# B&R Automation Studio project RobotComau (part 2)

#### Main.st
```iecst
PROGRAM _INIT
	(* Insert code here *)
	MpRecipeXml_0.MpLink := ADR(gRecipeXml);
	MpRecipeXml_0.Enable := TRUE;

	MpRecipeRegPar_0.MpLink := ADR(gRecipeXml);
	MpRecipeRegPar_0.Enable := TRUE;
	gAimPos;
	ScrewPosible := TRUE;
	ScrewWasherPosible := TRUE;
	WrenchPosible := TRUE;

	MpFileManagerUI_R(MpLink := ADR(gFileManagerUI_R), Enable :=1 , ErrorReset :=0 , UISetup :=MpFileMngSetup , UIConnect :=ADR(MpFileMngConnectR));
	MpFileMngConnectR.DeviceList.DeviceNames[0] := 'RecipeDir';

END_PROGRAM

PROGRAM _CYCLIC
	(* Insert code here *)

	IF clear THEN

		FOR i := 0 TO 13 BY 1 DO
		gAimPos[i] :=0 ;
		END_FOR;
		ScrewPosible := TRUE;
		ScrewWasherPosible := TRUE;
		WrenchPosible := TRUE;
	END_IF

	FOR i := 0 TO 13 BY 1 DO

		IF gAimPos[i]  = 1 THEN
			ScrewPosible := FALSE;
		END_IF
		IF gAimPos[i]  = 2 THEN
			ScrewWasherPosible := FALSE;
		END_IF
		IF gAimPos[i]  = 3 THEN
			ScrewPosible := FALSE;
			ScrewWasherPosible := FALSE;
		END_IF
		IF gAimPos[i]  = 4 THEN
			WrenchPosible := FALSE;
		END_IF
		IF gAimPos[i]  = 5 THEN
			WrenchPosible := FALSE;
			ScrewPosible := FALSE;
		END_IF
		IF gAimPos[i]  = 6 THEN
			WrenchPosible := FALSE;
			ScrewWasherPosible := FALSE;
		END_IF
		IF gAimPos[i]  = 7 THEN
			WrenchPosible := FALSE;
			ScrewPosible := FALSE;
			ScrewWasherPosible := FALSE;
		END_IF

	END_FOR;

	MpRecipeXml_0();
	MpRecipeXml_0.DeviceName := ADR('RecipeDir');
	MpRecipeRegPar_0();
	MpRecipeRegPar_0.PVName := ADR('gAimPos');

	MpRecipeXml_0.FileName := ADR(name);

	MpFileManagerUI_R();
	tabInfo.NumberOfElements := 0;

	IF MpFileMngConnectR.MessageBox.Type = mpFILE_MSG_OK THEN
		messageType := 'OK';
	ELSIF MpFileMngConnectR.MessageBox.Type = mpFILE_MSG_CONFIRM_DELETE THEN
		messageType := 'DELETE';
	ELSIF MpFileMngConnectR.MessageBox.Type = mpFILE_MSG_CONFIRM_OVERWRITE THEN
		messageType := 'OVERWRITE';
	ELSIF MpFileMngConnectR.MessageBox.Type = mpFILE_MSG_BUSY THEN
		messageType := 'BUSY';
	END_IF

	FOR iFile := 0 TO 49 BY 1 DO
		(* create arrays with file properties *)

		IF tabInfo.NumberOfElements >= iFile THEN
			brsmemcpy(ADR(tabInfo.Name[iFile]), ADR(MpFileMngConnectR.File.List.Items[iFile].Name), SIZEOF(tabInfo.Name[iFile]));
			brsmemcpy(ADR(tabInfo.Size[iFile]), ADR(MpFileMngConnectR.File.List.Items[iFile].Size), SIZEOF(tabInfo.Size[iFile]));
			brsmemcpy(ADR(tabInfo.Type[iFile]), ADR(MpFileMngConnectR.File.List.Items[iFile].ItemType), SIZEOF(tabInfo.Type[iFile]));
			brsmemcpy(ADR(tabInfo.LastModified[iFile]), ADR(MpFileMngConnectR.File.List.Items[iFile].LastModified), SIZEOF(tabInfo.LastModified[iFile]));
		END_IF

		IF tabInfo.SelectedRow = iFile THEN
			MpFileMngConnectR.File.List.Items[iFile].IsSelected := TRUE;
			name2 := MpFileMngConnectR.File.List.Items[iFile].Name;
		END_IF
		(* numbers of elements in the table *)
		IF tabInfo.Type[iFile] <> mpFILE_ITEM_TYPE_NONE THEN
			//			tabInfo.NumberOfElements := iFile;
			tabInfo.NumberOfElements := tabInfo.NumberOfElements + 1;
		END_IF
	END_FOR

	tableShowLimit := tabInfo.NumberOfElements - 1;
	tableConfig := '{"specRows": [ {"from":0, "to":';
	brsitoa(tableShowLimit,ADR(tempString));
	brsstrcat(ADR(tableConfig),ADR(tempString));
	brsstrcat(ADR(tableConfig),ADR(', "visible":true}, {"from":'));
	brsitoa(tabInfo.NumberOfElements,ADR(tempString));
	brsstrcat(ADR(tableConfig),ADR(tempString));
	brsstrcat(ADR(tableConfig),ADR(', "to":49, "visible":false}]}'));

	IF PriorytetS = 1 THEN
		Index[0] := 1;
	ELSIF PriorytetSW = 1 THEN
		Index[0] := 2;
	ELSIF PriorytetW = 1 THEN
		Index[0] := 4;
	END_IF

	IF PriorytetS = 2 THEN
		Index[1] := 1;
	ELSIF PriorytetSW = 2 THEN
		Index[1] := 2;
	ELSIF PriorytetW = 2 THEN
		Index[1] := 4;
	END_IF

	IF PriorytetS = 3 THEN
		Index[2] := 1;
	ELSIF PriorytetSW = 3 THEN
		Index[2] := 2;
	ELSIF PriorytetW = 3 THEN
		Index[2] := 4;
	END_IF

	IF PriorytetS = PriorytetSW OR PriorytetS = PriorytetW OR PriorytetSW = PriorytetW OR
		PriorytetS = 0 OR PriorytetSW = 0 OR PriorytetW = 0
		THEN
		Index[0] := 1;
		Index[1] := 2;
		Index[2] := 4;
	END_IF

END_PROGRAM

PROGRAM _EXIT
	(* Insert code here *)

END_PROGRAM
```

### Types.typ
```iecst
TYPE
	Step_typ :
		(
		ROBOTCTRL_DISABLED,
		ROBOTCTRL_POWER,
		ROBOTCTRL_WAIT_POWER,
		ROBOTCTRL_HOME,
		ROBOTCTRL_WAIT_HOME,
		ROBOTCTRL_READY,
		ROBOTCTRL_CALCULATE,
		ROBOTCTRL_CHECK,
		ROBOTCTRL_CALCULATE_P1,
		ROBOTCTRL_CALCULATE_P2,
		ROBOTCTRL_IS_MOVE_NEEDED,
		ROBOTCTRL_MOVE,
		ROBOTCTRL_ERROR_WRONG_AIM,
		ROBOTCTRL_ERROR,
		ROBOTCTRL_STOP,
		ROBOTCTRL_INTERRUPT,
		ROBOTCTRL_INTERRUPTING,
		ROBOTCTRL_CONTINUE,
		ROBOTCTRL_POWER_OFF,
		ROBOTCTRL_COMPLITE,
		ROBOTCTRL_SWAP,
		ROBOTCTRL_SWAP_MOVE,
		ROBOTCTRL_DEMO
		);
END_TYPE
```

### Variables.var
```iecst
VAR
	AimIsGood : BOOL := FALSE;
	cartezianVSjog : BOOL; (*Wybór miedzy sterowaniem we wspólrzednych wewnetrznych - 0 / zewnętrznych - 1 *)
	cmdContinue : BOOL;
	cmdInterrupt : BOOL;
	Demo : INT;
	DemoAimPos : ARRAY[0..13] OF INT; (*(DEMO) Aim poses used in demo *)
	DemoIndex : ARRAY[0..2] OF INT := [1,2,4]; (*(DEMO) Order Of movess*)
	diAck : BOOL; (*(IN AUTO)Resets of Vision system error*)
	diAuto : BOOL; (*Enables Auto mode*)
	diExecute : BOOL; (*(IN AUTO) Starts moving proedure *)
	diManual : BOOL; (*Enables manual mode*)
	diReset : BOOL; (*(IN AUTO)  Resets the procedure *)
	diSemiAuto : BOOL; (*Enables semiAuto mode*)
	diStart : BOOL; (*(IN AUTO) Sets robot ready *)
	diStop : BOOL; (*(IN AUTO) stops the procedure *)
	HelpfulInt : USINT; (*(SWAP) int that helps with assigning values *)
END_VAR
VAR CONSTANT
	IndexSize : INT := 3; (*Amount of diffrent objects *)
END_VAR
VAR
	MpRoboArm6Axis_0 : MpRoboArm6Axis; (*Robot *)
	P1P2_Ok : BOOL := FALSE; (*flag that shows if P1 and P2 was assigned*)
	PackML_State : STRING[80];
	RoboParameters : MpRoboArm6AxisParType; (*Robot Parameters*)
END_VAR
VAR CONSTANT
	SizeOfArray : INT := 13; (*(x+1)  amount of possible pleaces to move objects *)
END_VAR
VAR
	Step : {REDUND_UNREPLICABLE} Step_typ := (0); (*state robot *)
	Step_State : STRING[80];
	VelocityQ : REAL;
	VelocityQ1 : REAL; (*Przypisanie predkosci do parametru 1 w zależnosci od wyboru wspólrzednych*)
	VelocityQ2 : REAL; (*Przypisanie predkosci do parametru 2 w zależnosci od wyboru wspólrzednych*)
	VelocityQ3 : REAL; (*Przypisanie predkosci do parametru 3 w zależnosci od wyboru wspólrzednych*)
	VelocityQ4 : REAL; (*Przypisanie predkosci do parametru 4 w zależnosci od wyboru wspólrzednych*)
	VelocityQ5 : REAL; (*Przypisanie predkosci do parametru 5 w zależnosci od wyboru wspólrzednych*)
	VelocityQ6 : REAL; (*Przypisanie predkosci do parametru 6 w zależnosci od wyboru wspólrzednych*)
	VisionCalcDone : BOOL;
	SwapStep : USINT := 0; (*(SWAP) used in swap procedure *)
	x : INT := 0;
	VelocityQQ : REAL;
END_VAR
```

### Program Logical/Robot/PackML/PackML_Auto

#### Variables.var
```iecst
VAR
	NotFirstFlag : BOOL;
END_VAR
```

#### Aborted.st
```iecst
ACTION Aborted:

	IF MpPackMLStateIsActive(gPackMLCore,
		mpPACKML_STATE_ABORTED,
		1) THEN

		PackML_State := 'ABORTED';
		MpRoboArm6Axis_0.Power := FALSE;

		IF MpRoboArm6Axis_0.ErrorReset THEN
			MpPackMLStateComplete(gPackMLCore, 1);

			MpPackMLMode_Auto.Clear := 1;

		END_IF;
	END_IF

END_ACTION
```

#### Aborting.st
```iecst
ACTION Aborting:

	IF MpPackMLStateIsActive(gPackMLCore,
		mpPACKML_STATE_ABORTING,
		1) THEN

		MpPackMLMode_Auto.Abort := 0;

		PackML_State := 'ABORTING';
		MpRoboArm6Axis_0.Power := FALSE;

		IF NOT MpRoboArm6Axis_0.PowerOn THEN
			MpPackMLStateComplete(gPackMLCore, 1);

//			Step := ROBOTCTRL_POWER_OFF;
//			Step_State := 'POWER_OFF';

		END_IF;
	END_IF

END_ACTION
```

#### Clearing.st
```iecst
ACTION Clearing:

	IF MpPackMLStateIsActive(gPackMLCore,
		mpPACKML_STATE_CLEARING,
		1) THEN

		MpPackMLMode_Auto.Clear := 0;
		PackML_State := 'CLEARING';

		IF NOT MpRoboArm6Axis_0.Error THEN
			MpPackMLStateComplete(gPackMLCore, 1);

		END_IF;
	END_IF
END_ACTION
```

#### Complete.st
```iecst
ACTION Complete:
	IF MpPackMLStateIsActive(gPackMLCore,
		mpPACKML_STATE_COMPLETE,
		1) THEN

		PackML_State := 'COMPLETE';
		gCompliteFlag:=TRUE;
		//MpPackMLMode_Auto.Stop := 1;

		IF diReset THEN
			MpPackMLStateComplete(gPackMLCore, 1);
			MpPackMLMode_Auto.Reset := 1;
			Step := ROBOTCTRL_POWER;

			//			Step_State := 'POWER';

			END_IF;
	END_IF

END_ACTION
```

#### Completing.st
```iecst
ACTION Completing:
	IF MpPackMLStateIsActive(gPackMLCore,
		mpPACKML_STATE_COMPLETING,
		1) THEN
			PackML_State := 'COMPLETING';
		emptyPos:=0;
			MpPackMLStateComplete(gPackMLCore, 1);

	END_IF

END_ACTION
```

#### Execute.st
```iecst
//   General conception of this code
//  assainging binary values to each object
//	screw      -001 - 1
//  screw pad  -010 - 2
//  wrench     -100 - 4
//  therefore we can assing to gAimPose table values from 0-7 ( sum must equal 7) in order to
//  easly differentiate what kind of object we need to move into aim pose.
//  for example if we see 6 -> 110 we know that we have to move screw pad and wrench to this pose
//
//  order of moves is defined by order of numbers in Index

ACTION Execute:
	IF MpPackMLStateIsActive(gPackMLCore,
		mpPACKML_STATE_EXECUTE,
		1) THEN

		PackML_State := 'EXECUTE';

		CASE Step OF

			ROBOTCTRL_CALCULATE:
				//Reseting buffor
				//blocks which can be used as buffor
				FOR x:=0 TO SizeOfArray DO
					IF  gActPos[x]=0 THEN
						gSwapEnable[x]:=FALSE;
					ELSE
						gSwapEnable[x]:=TRUE;
					END_IF;
				END_FOR;

				IF diDemo THEN
					IF NOT NotFirstFlag THEN
						FOR x:=0 TO SizeOfArray DO
							gDemoActPos[x]:=gActPos[x];
						END_FOR;
					END_IF;

					FOR x:=0 TO SizeOfArray DO
						IF  gDemoActPos[x]=0 AND gIsPosGood[x] THEN
							gPosBuffor[x]:=TRUE;
						ELSE
							gPosBuffor[x]:=FALSE;
						END_IF;
					END_FOR;
				ELSE
					FOR x:=0 TO SizeOfArray DO
						IF  gActPos[x]=0 AND gIsPosGood[x] THEN
							gPosBuffor[x]:=TRUE;
						ELSE
							gPosBuffor[x]:=FALSE;
						END_IF;
					END_FOR;

				END_IF;

				IF diDemo AND NOT P1P2_Ok AND y=0 THEN
					CASE Demo OF

						0:
							DemoY:=0;
							DemoIndex[0]:=1;
							DemoIndex[1]:=2;
							DemoIndex[2]:=4;
							FOR x:=0 TO SizeOfArray DO
								IF DemoY <IndexSize THEN
									IF gPosBuffor[x] THEN
										DemoAimPos[x]:=DemoIndex[DemoY];
										DemoY:=DemoY+1;
									ELSE
										DemoAimPos[x]:=0;

									END_IF;
								ELSE
									DemoAimPos[x]:=0;
								END_IF;
							END_FOR;
							Step:=ROBOTCTRL_CALCULATE_P1;
							Demo:=1;

						1:

							DemoY:=0;
							DemoIndex[0]:=2;
							DemoIndex[1]:=1;
							DemoIndex[2]:=4;
							FOR x:=SizeOfArray TO 0 BY -1 DO
								IF DemoY <IndexSize THEN
									IF gPosBuffor[x] THEN
										DemoAimPos[x]:=DemoIndex[DemoY];
										DemoY:=DemoY+1;
									ELSE
										DemoAimPos[x]:=0;

									END_IF;
								ELSE
									DemoAimPos[x]:=0;
								END_IF;

							END_FOR;
							Step:=ROBOTCTRL_CALCULATE_P1;
							Demo:=2;

						2:

							DemoY:=0;
							DemoIndex[0]:=4;
							DemoIndex[1]:=2;
							DemoIndex[2]:=1;
							FOR x:=0 TO SizeOfArray DO
								IF DemoY <IndexSize THEN
									IF gPosBuffor[x] THEN
										DemoAimPos[x]:=DemoIndex[DemoY];
										DemoY:=DemoY+1;
									ELSE
										DemoAimPos[x]:=0;

									END_IF;
								ELSE
									DemoAimPos[x]:=0;
								END_IF;
							END_FOR;
							Step:=ROBOTCTRL_CALCULATE_P1;
							Demo:=3;

						3:

							DemoY:=0;
							DemoIndex[0]:=1;
							DemoIndex[1]:=4;
							DemoIndex[2]:=2;
							FOR x:=SizeOfArray TO 0 BY -1 DO
								IF DemoY <IndexSize THEN
									IF gPosBuffor[x] THEN
										DemoAimPos[x]:=DemoIndex[DemoY];
										DemoY:=DemoY+1;
									ELSE
										DemoAimPos[x]:=0;

									END_IF;
								ELSE
									DemoAimPos[x]:=0;
								END_IF;
							END_FOR;
							Step:=ROBOTCTRL_CALCULATE_P1;
							Demo:=0;

					END_CASE;

				ELSIF	gSwapFlag THEN
					gSwapFlag:=FALSE;
					Step:=ROBOTCTRL_SWAP;
				ELSIF P1P2_Ok THEN
					Step:=ROBOTCTRL_IS_MOVE_NEEDED;
				ELSIF y<IndexSize THEN
					Step:=ROBOTCTRL_CALCULATE_P1;
				ELSE
					diStart:=FALSE;
					RoboParameters.ProgramName := 'HOME.st';
					MpRoboArm6Axis_0.MoveProgram:=1;
					IF MpRoboArm6Axis_0.MoveDone THEN
						MpRoboArm6Axis_0.MoveProgram:=FALSE;
						MpPackMLStateComplete(gPackMLCore, 1);
					END_IF

				END_IF;

			ROBOTCTRL_CALCULATE_P1:
				//assigning values to P1 and P1up

				IF diDemo THEN
					FOR x:=0  TO SizeOfArray DO
						IF gDemoActPos[x]=DemoIndex[y] THEN
							P1.Orient.Angle1:=gRobPos[x].Orient.Angle1;
							P1.Orient.Angle2:=gRobPos[x].Orient.Angle2;
							P1.Orient.Angle3:=gRobPos[x].Orient.Angle3;
							P1.Pos.X:=gRobPos[x].Pos.X;
							P1.Pos.Y:=gRobPos[x].Pos.Y;
							P1.Pos.Z:=gRobPos[x].Pos.Z;
							P1up.Orient.Angle1:=gRobPos[x].Orient.Angle1;
							P1up.Orient.Angle2:=gRobPos[x].Orient.Angle2;
							P1up.Orient.Angle3:=gRobPos[x].Orient.Angle3;
							P1up.Pos.X:=gRobPos[x].Pos.X;
							P1up.Pos.Y:=gRobPos[x].Pos.Y;
							P1up.Pos.Z:=gRobPos[x].Pos.Z+50;
						END_IF;
					END_FOR;
				ELSE
					FOR x:=0  TO SizeOfArray DO
						IF gActPos[x]=Index[y] THEN
							P1.Orient.Angle1:=gRobPos[x].Orient.Angle1;
							P1.Orient.Angle2:=gRobPos[x].Orient.Angle2;
							P1.Orient.Angle3:=gRobPos[x].Orient.Angle3;
							P1.Pos.X:=gRobPos[x].Pos.X;
							P1.Pos.Y:=gRobPos[x].Pos.Y;
							P1.Pos.Z:=gRobPos[x].Pos.Z;
							P1up.Orient.Angle1:=gRobPos[x].Orient.Angle1;
							P1up.Orient.Angle2:=gRobPos[x].Orient.Angle2;
							P1up.Orient.Angle3:=gRobPos[x].Orient.Angle3;
							P1up.Pos.X:=gRobPos[x].Pos.X;
							P1up.Pos.Y:=gRobPos[x].Pos.Y;
							P1up.Pos.Z:=gRobPos[x].Pos.Z+50;
						END_IF;
					END_FOR;
				END_IF;

				Step:=ROBOTCTRL_CALCULATE_P2;
				Step_State := 'CALCULATE_P2';

			ROBOTCTRL_CALCULATE_P2:
				IF diDemo THEN
					FOR x:=0 TO SizeOfArray DO
						//copig values
						gAimPos1[x]:=DemoAimPos[x];
					END_FOR;
					FOR x:=0 TO SizeOfArray DO
						//reseting maps
						Aim1[x]:=FALSE;
						Aim2[x]:=FALSE;
						Aim4[x]:=FALSE;
					END_FOR;
					//Creating maps conteining positions of each element
					//by substracting corresponding value of element
					//AND checing IF its greater OR equal TO zero
					FOR z:=0 TO IndexSize DO
						IF DemoIndex[z]=4 THEN
							FOR x:=0 TO SizeOfArray DO
								IF((gAimPos1[x]-4)>=0) THEN
									gAimPos1[x]:=gAimPos1[x]-4;
									Aim4[x]:=TRUE;
								END_IF;
							END_FOR;
						END_IF;
					END_FOR;

					FOR z:=0 TO IndexSize DO
						IF DemoIndex[z]=2 THEN
							FOR x:=0 TO SizeOfArray DO
								IF((gAimPos1[x]-2)>=0) THEN
									gAimPos1[x]:=gAimPos1[x]-2;
									Aim2[x]:=TRUE;
								END_IF;
							END_FOR;
						END_IF;
					END_FOR;

					FOR z:=0 TO IndexSize DO
						IF DemoIndex[z]=1 THEN
							FOR x:=0 TO SizeOfArray DO
								IF((gAimPos1[x]-1)>=0) THEN
									gAimPos1[x]:=gAimPos1[x]-1;
									Aim1[x]:=TRUE;
								END_IF;
							END_FOR;
						END_IF;
					END_FOR;

					IF DemoIndex[y]=4 THEN
						//moving in order defined in Index
						FOR x:=0  TO SizeOfArray DO
							IF Aim4[x] THEN
								P2.Orient.Angle1:=gRobPos[x].Orient.Angle1;
								P2.Orient.Angle2:=gRobPos[x].Orient.Angle2;
								P2.Orient.Angle3:=gRobPos[x].Orient.Angle3;
								P2.Pos.X:=gRobPos[x].Pos.X;
								P2.Pos.Y:=gRobPos[x].Pos.Y;
								P2.Pos.Z:=gRobPos[x].Pos.Z;
								P2up.Orient.Angle1:=gRobPos[x].Orient.Angle1;
								P2up.Orient.Angle2:=gRobPos[x].Orient.Angle2;
								P2up.Orient.Angle3:=gRobPos[x].Orient.Angle3;
								P2up.Pos.X:=gRobPos[x].Pos.X;
								P2up.Pos.Y:=gRobPos[x].Pos.Y;
								P2up.Pos.Z:=gRobPos[x].Pos.Z+50;

							END_IF;
						END_FOR;
					ELSIF DemoIndex[y]=2 THEN
						FOR x:=0  TO SizeOfArray DO
							IF Aim2[x] THEN
								P2.Orient.Angle1:=gRobPos[x].Orient.Angle1;
								P2.Orient.Angle2:=gRobPos[x].Orient.Angle2;
								P2.Orient.Angle3:=gRobPos[x].Orient.Angle3;
								P2.Pos.X:=gRobPos[x].Pos.X;
								P2.Pos.Y:=gRobPos[x].Pos.Y;
								P2.Pos.Z:=gRobPos[x].Pos.Z;
								P2up.Orient.Angle1:=gRobPos[x].Orient.Angle1;
								P2up.Orient.Angle2:=gRobPos[x].Orient.Angle2;
								P2up.Orient.Angle3:=gRobPos[x].Orient.Angle3;
								P2up.Pos.X:=gRobPos[x].Pos.X;
								P2up.Pos.Y:=gRobPos[x].Pos.Y;
								P2up.Pos.Z:=gRobPos[x].Pos.Z+50;

							END_IF;
						END_FOR;
					ELSIF DemoIndex[y]=1 THEN
						FOR x:=0  TO SizeOfArray DO
							IF Aim1[x] THEN
								P2.Orient.Angle1:=gRobPos[x].Orient.Angle1;
								P2.Orient.Angle2:=gRobPos[x].Orient.Angle2;
								P2.Orient.Angle3:=gRobPos[x].Orient.Angle3;
								P2.Pos.X:=gRobPos[x].Pos.X;
								P2.Pos.Y:=gRobPos[x].Pos.Y;
								P2.Pos.Z:=gRobPos[x].Pos.Z;
								P2up.Orient.Angle1:=gRobPos[x].Orient.Angle1;
								P2up.Orient.Angle2:=gRobPos[x].Orient.Angle2;
								P2up.Orient.Angle3:=gRobPos[x].Orient.Angle3;
								P2up.Pos.X:=gRobPos[x].Pos.X;
								P2up.Pos.Y:=gRobPos[x].Pos.Y;
								P2up.Pos.Z:=gRobPos[x].Pos.Z+50;

							END_IF;
						END_FOR;
					END_IF;
				ELSE
					FOR x:=0 TO SizeOfArray DO
						//copig values
						gAimPos1[x]:=gAimPos[x];
					END_FOR;
					FOR x:=0 TO SizeOfArray DO
						//reseting maps
						Aim1[x]:=FALSE;
						Aim2[x]:=FALSE;
						Aim4[x]:=FALSE;
					END_FOR;
					//Creating maps conteining positions of each element
					//by substracting corresponding value of element
					//AND checing IF its greater OR equal TO zero
					FOR z:=0 TO IndexSize DO
						IF Index[z]=4 THEN
							FOR x:=0 TO SizeOfArray DO
								IF((gAimPos1[x]-4)>=0) THEN
									gAimPos1[x]:=gAimPos1[x]-4;
									Aim4[x]:=TRUE;
								END_IF;
							END_FOR;
						END_IF;
					END_FOR;

					FOR z:=0 TO IndexSize DO
						IF Index[z]=2 THEN
							FOR x:=0 TO SizeOfArray DO
								IF((gAimPos1[x]-2)>=0) THEN
									gAimPos1[x]:=gAimPos1[x]-2;
									Aim2[x]:=TRUE;
								END_IF;
							END_FOR;
						END_IF;
					END_FOR;

					FOR z:=0 TO IndexSize DO
						IF Index[z]=1 THEN
							FOR x:=0 TO SizeOfArray DO
								IF((gAimPos1[x]-1)>=0) THEN
									gAimPos1[x]:=gAimPos1[x]-1;
									Aim1[x]:=TRUE;
								END_IF;
							END_FOR;
						END_IF;
					END_FOR;

					//assigning values to P2 and P2up
					IF Index[y]=4 THEN
						//moving in order defined in Index
						FOR x:=0  TO SizeOfArray DO
							IF Aim4[x] THEN
								P2.Orient.Angle1:=gRobPos[x].Orient.Angle1;
								P2.Orient.Angle2:=gRobPos[x].Orient.Angle2;
								P2.Orient.Angle3:=gRobPos[x].Orient.Angle3;
								P2.Pos.X:=gRobPos[x].Pos.X;
								P2.Pos.Y:=gRobPos[x].Pos.Y;
								P2.Pos.Z:=gRobPos[x].Pos.Z;
								P2up.Orient.Angle1:=gRobPos[x].Orient.Angle1;
								P2up.Orient.Angle2:=gRobPos[x].Orient.Angle2;
								P2up.Orient.Angle3:=gRobPos[x].Orient.Angle3;
								P2up.Pos.X:=gRobPos[x].Pos.X;
								P2up.Pos.Y:=gRobPos[x].Pos.Y;
								P2up.Pos.Z:=gRobPos[x].Pos.Z+50;
							END_IF;
						END_FOR;
					ELSIF Index[y]=2 THEN
						FOR x:=0  TO SizeOfArray DO
							IF Aim2[x] THEN
								P2.Orient.Angle1:=gRobPos[x].Orient.Angle1;
								P2.Orient.Angle2:=gRobPos[x].Orient.Angle2;
								P2.Orient.Angle3:=gRobPos[x].Orient.Angle3;
								P2.Pos.X:=gRobPos[x].Pos.X;
								P2.Pos.Y:=gRobPos[x].Pos.Y;
								P2.Pos.Z:=gRobPos[x].Pos.Z;
								P2up.Orient.Angle1:=gRobPos[x].Orient.Angle1;
								P2up.Orient.Angle2:=gRobPos[x].Orient.Angle2;
								P2up.Orient.Angle3:=gRobPos[x].Orient.Angle3;
								P2up.Pos.X:=gRobPos[x].Pos.X;
								P2up.Pos.Y:=gRobPos[x].Pos.Y;
								P2up.Pos.Z:=gRobPos[x].Pos.Z+50;
							END_IF;
						END_FOR;
					ELSIF Index[y]=1 THEN
						FOR x:=0  TO SizeOfArray DO
							IF Aim1[x] THEN
								P2.Orient.Angle1:=gRobPos[x].Orient.Angle1;
								P2.Orient.Angle2:=gRobPos[x].Orient.Angle2;
								P2.Orient.Angle3:=gRobPos[x].Orient.Angle3;
								P2.Pos.X:=gRobPos[x].Pos.X;
								P2.Pos.Y:=gRobPos[x].Pos.Y;
								P2.Pos.Z:=gRobPos[x].Pos.Z;
								P2up.Orient.Angle1:=gRobPos[x].Orient.Angle1;
								P2up.Orient.Angle2:=gRobPos[x].Orient.Angle2;
								P2up.Orient.Angle3:=gRobPos[x].Orient.Angle3;
								P2up.Pos.X:=gRobPos[x].Pos.X;
								P2up.Pos.Y:=gRobPos[x].Pos.Y;
								P2up.Pos.Z:=gRobPos[x].Pos.Z+50;
							END_IF;
						END_FOR;
					END_IF;
				END_IF;

				P1P2_Ok:=1; // this flag means that new P1 and new P2 have been assigned
				Step:=ROBOTCTRL_CALCULATE;

			ROBOTCTRL_IS_MOVE_NEEDED:
				//checking if actual and aim positions are not the same
				IF P1.Orient.Angle1=P2.Orient.Angle1 AND P1.Pos.X=P2.Pos.X AND P1.Orient.Angle2=P2.Orient.Angle2 AND P1.Pos.Y=P2.Pos.Y AND P1.Orient.Angle3=P2.Orient.Angle3 AND P1.Pos.Z=P2.Pos.Z THEN
					y:=y+1; // index of next object
					P1P2_Ok:=0; // ready to assign new values to p1 p1up p2 p2up
					Step:=ROBOTCTRL_CALCULATE; // next assigning procedure with new object
					Step_State := 'CALCULATE';
				ELSE
					Step_State := 'MOVE';
					Step:=ROBOTCTRL_MOVE;   // going to move command
				END_IF;

			ROBOTCTRL_MOVE:
				IF cmdInterrupt OR MpRoboArm6Axis_0.MoveInterrupted THEN
					cmdInterrupt := FALSE;
					Step:=ROBOTCTRL_INTERRUPT;
					Step_State := 'INTERRUPT';
					MpPackMLMode_Auto.Hold := 1;
				END_IF;

				//executing move procedure
				MpRoboArm6Axis_0.MoveProgram:=1;
				IF MpRoboArm6Axis_0.MoveDone THEN
					//restarting assigning procedure with new object after finishing move
					MpRoboArm6Axis_0.MoveProgram:=0;
					y:=y+1;
					IF diDemo AND y=IndexSize THEN
						FOR x:=0 TO SizeOfArray DO
							gDemoActPos[x]:=DemoAimPos[x];
						END_FOR;
						y:=0;
						NotFirstFlag:=TRUE;

					END_IF
					P1P2_Ok:=0;
					Step:=ROBOTCTRL_CALCULATE;
					Step_State := 'CALCULATE';

				END_IF
				//////////////////////////////////////////////////////////////////////////////////////////////////////////////////////////
				///////////////////////////////////////////////////SWAP///////////////////////////////////////////////////////////////////
				//////////////////////////////////////////////////////////////////////////////////////////////////////////////////////////
			ROBOTCTRL_SWAP:
				gSwapFlag:=FALSE;
				HelpfulInt:=0;
				FOR x:=0 TO SizeOfArray DO
					//swap map can have only 2 values that are TRUE those coordinates are going to be swaped
					IF gSwapMap[x] THEN
						gSwapPoses[HelpfulInt].Orient.Angle1:=gRobPos[x].Orient.Angle1;
						gSwapPoses[HelpfulInt].Orient.Angle2:=gRobPos[x].Orient.Angle2;
						gSwapPoses[HelpfulInt].Orient.Angle3:=gRobPos[x].Orient.Angle3;
						gSwapPoses[HelpfulInt].Pos.X:=gRobPos[x].Pos.X;
						gSwapPoses[HelpfulInt].Pos.Y:=gRobPos[x].Pos.Y;
						gSwapPoses[HelpfulInt].Pos.Z:=gRobPos[x].Pos.Z;
						HelpfulInt:=HelpfulInt + 1;
					END_IF
				END_FOR;
				//gSwapMap should only have 2 values equal to TRUE therefore HelpfulInt should equal to 2
				//but just in case it is better to assign 2 to HelpfulInt
				HelpfulInt:=2;

				FOR x:=0 TO SizeOfArray DO
					IF gPosBuffor[x] THEN
						gSwapPoses[HelpfulInt].Orient.Angle1:=gRobPos[x].Orient.Angle1;
						gSwapPoses[HelpfulInt].Orient.Angle2:=gRobPos[x].Orient.Angle2;
						gSwapPoses[HelpfulInt].Orient.Angle3:=gRobPos[x].Orient.Angle3;
						gSwapPoses[HelpfulInt].Pos.X:=gRobPos[x].Pos.X;
						gSwapPoses[HelpfulInt].Pos.Y:=gRobPos[x].Pos.Y;
						gSwapPoses[HelpfulInt].Pos.Z:=gRobPos[x].Pos.Z;
						EXIT;
					END_IF
				END_FOR;

				FOR x:=0 TO SizeOfArray DO
					gSwapMap[x]:=FALSE;
				END_FOR;
				y:=0;
				Step:=ROBOTCTRL_SWAP_MOVE;

			ROBOTCTRL_SWAP_MOVE:

				CASE SwapStep OF
					0:
						//First move
						///////////////////////P1
						P1.Orient.Angle1:=gSwapPoses[0].Orient.Angle1;
						P1.Orient.Angle2:=gSwapPoses[0].Orient.Angle2;
						P1.Orient.Angle3:=gSwapPoses[0].Orient.Angle3;
						P1.Pos.X:=gSwapPoses[0].Pos.X;
						P1.Pos.Y:=gSwapPoses[0].Pos.Y;
						P1.Pos.Z:=gSwapPoses[0].Pos.Z;
						P1up.Orient.Angle1:=gSwapPoses[0].Orient.Angle1;
						P1up.Orient.Angle2:=gSwapPoses[0].Orient.Angle2;
						P1up.Orient.Angle3:=gSwapPoses[0].Orient.Angle3;
						P1up.Pos.X:=gSwapPoses[0].Pos.X;
						P1up.Pos.Y:=gSwapPoses[0].Pos.Y;
						P1up.Pos.Z:=gSwapPoses[0].Pos.Z+50;
						///////////////////////P2
						P2.Orient.Angle1:=gSwapPoses[2].Orient.Angle1;
						P2.Orient.Angle2:=gSwapPoses[2].Orient.Angle2;
						P2.Orient.Angle3:=gSwapPoses[2].Orient.Angle3;
						P2.Pos.X:=gSwapPoses[2].Pos.X;
						P2.Pos.Y:=gSwapPoses[2].Pos.Y;
						P2.Pos.Z:=gSwapPoses[2].Pos.Z;
						P2up.Orient.Angle1:=gSwapPoses[2].Orient.Angle1;
						P2up.Orient.Angle2:=gSwapPoses[2].Orient.Angle2;
						P2up.Orient.Angle3:=gSwapPoses[2].Orient.Angle3;
						P2up.Pos.X:=gSwapPoses[2].Pos.X;
						P2up.Pos.Y:=gSwapPoses[2].Pos.Y;
						P2up.Pos.Z:=gSwapPoses[2].Pos.Z+50;
						RoboParameters.ProgramName := 'Robotic.st';
						//////////////////////// command execute
						MpRoboArm6Axis_0.MoveProgram:=1;
						IF MpRoboArm6Axis_0.MoveDone  THEN
							MpRoboArm6Axis_0.MoveProgram:=0;
							SwapStep:=1;
						END_IF;
					1:
						//second move
						///////////////////////P1
						P1.Orient.Angle1:=gSwapPoses[1].Orient.Angle1;
						P1.Orient.Angle2:=gSwapPoses[1].Orient.Angle2;
						P1.Orient.Angle3:=gSwapPoses[1].Orient.Angle3;
						P1.Pos.X:=gSwapPoses[1].Pos.X;
						P1.Pos.Y:=gSwapPoses[1].Pos.Y;
						P1.Pos.Z:=gSwapPoses[1].Pos.Z;
						P1up.Orient.Angle1:=gSwapPoses[1].Orient.Angle1;
						P1up.Orient.Angle2:=gSwapPoses[1].Orient.Angle2;
						P1up.Orient.Angle3:=gSwapPoses[1].Orient.Angle3;
						P1up.Pos.X:=gSwapPoses[1].Pos.X;
						P1up.Pos.Y:=gSwapPoses[1].Pos.Y;
						P1up.Pos.Z:=gSwapPoses[1].Pos.Z+50;
						///////////////////////P2
						P2.Orient.Angle1:=gSwapPoses[0].Orient.Angle1;
						P2.Orient.Angle2:=gSwapPoses[0].Orient.Angle2;
						P2.Orient.Angle3:=gSwapPoses[0].Orient.Angle3;
						P2.Pos.X:=gSwapPoses[0].Pos.X;
						P2.Pos.Y:=gSwapPoses[0].Pos.Y;
						P2.Pos.Z:=gSwapPoses[0].Pos.Z;
						P2up.Orient.Angle1:=gSwapPoses[0].Orient.Angle1;
						P2up.Orient.Angle2:=gSwapPoses[0].Orient.Angle2;
						P2up.Orient.Angle3:=gSwapPoses[0].Orient.Angle3;
						P2up.Pos.X:=gSwapPoses[0].Pos.X;
						P2up.Pos.Y:=gSwapPoses[0].Pos.Y;
						P2up.Pos.Z:=gSwapPoses[0].Pos.Z+50;
						y:=1;
						RoboParameters.ProgramName := 'Robotic.st';
						//////////////////////// command execute
						MpRoboArm6Axis_0.MoveProgram:=1;
						IF MpRoboArm6Axis_0.MoveDone   THEN
							MpRoboArm6Axis_0.MoveProgram:=0;
							SwapStep:=2;
						END_IF;

					2:
						//third move
						///////////////////////P1
						P1.Orient.Angle1:=gSwapPoses[2].Orient.Angle1;
						P1.Orient.Angle2:=gSwapPoses[2].Orient.Angle2;
						P1.Orient.Angle3:=gSwapPoses[2].Orient.Angle3;
						P1.Pos.X:=gSwapPoses[2].Pos.X;
						P1.Pos.Y:=gSwapPoses[2].Pos.Y;
						P1.Pos.Z:=gSwapPoses[2].Pos.Z;
						P1up.Orient.Angle1:=gSwapPoses[2].Orient.Angle1;
						P1up.Orient.Angle2:=gSwapPoses[2].Orient.Angle2;
						P1up.Orient.Angle3:=gSwapPoses[2].Orient.Angle3;
						P1up.Pos.X:=gSwapPoses[2].Pos.X;
						P1up.Pos.Y:=gSwapPoses[2].Pos.Y;
						P1up.Pos.Z:=gSwapPoses[2].Pos.Z+50;
						///////////////////////P2
						P2.Orient.Angle1:=gSwapPoses[1].Orient.Angle1;
						P2.Orient.Angle2:=gSwapPoses[1].Orient.Angle2;
						P2.Orient.Angle3:=gSwapPoses[1].Orient.Angle3;
						P2.Pos.X:=gSwapPoses[1].Pos.X;
						P2.Pos.Y:=gSwapPoses[1].Pos.Y;
						P2.Pos.Z:=gSwapPoses[1].Pos.Z;
						P2up.Orient.Angle1:=gSwapPoses[1].Orient.Angle1;
						P2up.Orient.Angle2:=gSwapPoses[1].Orient.Angle2;
						P2up.Orient.Angle3:=gSwapPoses[1].Orient.Angle3;
						P2up.Pos.X:=gSwapPoses[1].Pos.X;
						P2up.Pos.Y:=gSwapPoses[1].Pos.Y;
						P2up.Pos.Z:=gSwapPoses[1].Pos.Z+50;
						y:=2;
						RoboParameters.ProgramName := 'Robotic.st';
						MpRoboArm6Axis_0.MoveProgram:=1;
						IF MpRoboArm6Axis_0.MoveDone   THEN
							MpRoboArm6Axis_0.MoveProgram:=0;
							SwapStep:=3;
						END_IF;

					3:
						SwapStep:=0;
						MpPackMLStateComplete(gPackMLCore, 1);

				END_CASE ;

		END_CASE;

	END_IF;

				END_ACTION
```

#### Held.st
```iecst
ACTION Held:

	IF MpPackMLStateIsActive(gPackMLCore,
		mpPACKML_STATE_HELD,
		1) THEN

		PackML_State := 'HELD';

		IF cmdContinue THEN
			cmdContinue:=FALSE;
			MpRoboArm6Axis_0.Interrupt:=FALSE;
//			Step:=ROBOTCTRL_CONTINUE;
//			Step_State := 'CONTINUE';
			MpPackMLMode_Auto.Unhold := 1;
		END_IF
	END_IF

END_ACTION
```

#### Holding.st
```iecst
ACTION Holding:

	IF MpPackMLStateIsActive(gPackMLCore,
		mpPACKML_STATE_HOLDING,
		1) THEN

		PackML_State := 'HOLDING';

		MpRoboArm6Axis_0.Interrupt:=TRUE;
		IF MpRoboArm6Axis_0.MoveInterrupted THEN
//			Step:=ROBOTCTRL_INTERRUPTING;
//			Step_State := 'INTERRUPTING';
			MpPackMLStateComplete(gPackMLCore, 1);
		END_IF
	END_IF

END_ACTION
```

#### Idle.st
```iecst
ACTION Idle:

	IF MpPackMLStateIsActive(gPackMLCore,
		mpPACKML_STATE_IDLE,
		1) THEN

		MpPackMLMode_Auto.Reset := 0;

		PackML_State := 'IDLE';

		//		CASE Step OF
		//			ROBOTCTRL_READY:
		MpRoboArm6Axis_0.MoveProgram := 0;

		FOR x:=0 TO SizeOfArray DO
			IF  gActPos[x]=0 THEN
				gSwapEnable[x]:=FALSE;
			ELSE
				gSwapEnable[x]:=TRUE;
			END_IF;
		END_FOR;

		IF NOT(MpRoboArm6Axis_0.PowerOn) THEN
			//					Step := ROBOTCTRL_DISABLED;
			//					Step_State := 'DISABLED';
			MpPackMLMode_Auto.Stop := TRUE;
		END_IF;

		IF diStart  THEN // diStart is active robot starts procedure
			diStart := FALSE;
			MpPackMLMode_Auto.Start := TRUE;
			Step := ROBOTCTRL_CHECK;
			Step_State := 'CHECK';
		END_IF;

		//		END_CASE;

	END_IF

END_ACTION
```

#### Main.st
```iecst
PROGRAM _INIT
	RestorePos;
	MpRoboArm6Axis_0.Enable := TRUE;

	MpRoboArm6Axis_0.Interrupt := 0;
	MpRoboArm6Axis_0.Continue := 0;
	gWait;
	MpRoboArm6Axis_0.Override  := 100.0;
	RoboParameters.CoordSystem := 0;
	RoboParameters.Velocity := 100;
	RoboParameters.Acceleration := 1000;
	RoboParameters.Deceleration := 1000;
	RoboParameters.ProgramName := 'Robotic.st';

END_PROGRAM

PROGRAM _CYCLIC
	Starting;
	Idle;
	Stopping;
	Resetting;
	Execute;
	Completing;
	Complete;
	Stopped;
	Holding;
	Held;
	Unhold;
	Aborted;
	Aborting;
	Clearing;

	P2up;
	P2 ;
	P1up ;
	P1 ;
	P0;
	HOME;
	PZ;
	A;
	doMagnet;
	MaxSpeed;
	LowSpeed;

	IF diAck THEN
		doVisError:=FALSE;

	END_IF;

	//throwing error
	IF MpRoboArm6Axis_0.Error THEN
		//		Step := ROBOTCTRL_ERROR;
		MpPackMLMode_Auto.Abort := TRUE;
		//		Step_State := 'ERROR';
	END_IF;

	IF diStop THEN
		MpRoboArm6Axis_0.Power := 0;
		MpPackMLMode_Auto.Stop := 1;
		//		Step := ROBOTCTRL_POWER_OFF;
		//		Step_State := 'POWER_OFF';
	END_IF

	MpPackMLCore_0;
	MpPackMLMode_Auto;

	diStop;
	diStart;
	diReset;
	diExecute;
	cmdContinue;

	diAuto;
	diSemiAuto;
	diManual;

	MpRoboArm6Axis_0.MpLink     := ADR(gAxesGroup_Racer3_1);
	MpRoboArm6Axis_0.Parameters := ADR(RoboParameters);
	MpRoboArm6Axis_0.Override := 100.0;
	MpRoboArm6Axis_0.Enable := TRUE;
	MpRoboArm6Axis_0();

END_PROGRAM

PROGRAM _EXIT

END_PROGRAM
```

#### Resetting.st
```iecst
ACTION Resetting:

	IF MpPackMLStateIsActive(gPackMLCore,
		mpPACKML_STATE_RESETTING,
		1) THEN
		MpPackMLMode_Auto.Reset := 0;
		MpPackMLMode_Auto.Stop := 0;
		PackML_State := 'RESETTING';
		gCompliteFlag:=FALSE;
		y := 0;
		NotFirstFlag:=FALSE;
		Camera_0.ImageAcq := Camera_0.Ready;
		emptyPos:=0;
		IF NOT MpRoboArm6Axis_0.PowerOn THEN
			MpPackMLMode_Auto.Stop := 1;
		END_IF

		FOR x:=0 TO 5 DO
			FOR y:=0 TO 17 DO
				IF  RestorePos[x].Data[y]=0 THEN
				emptyPos:=emptyPos+1;
				END_IF
			END_FOR;
		END_FOR;

		CASE Step OF
			ROBOTCTRL_POWER:

				IF MpRoboArm6Axis_0.Info.ReadyToPowerOn THEN
					MpRoboArm6Axis_0.Power := TRUE;
					Step := ROBOTCTRL_WAIT_POWER;
					Step_State := 'WAIT_POWER';
				END_IF;

			ROBOTCTRL_WAIT_POWER:
				IF MpRoboArm6Axis_0.PowerOn THEN
					Step := ROBOTCTRL_HOME;
					Step_State := 'HOME';
				END_IF;

			ROBOTCTRL_HOME:
				MpRoboArm6Axis_0.Home := TRUE;
				Step := ROBOTCTRL_WAIT_HOME;
				Step_State := 'WAIT_HOME';

			ROBOTCTRL_WAIT_HOME:
				IF MpRoboArm6Axis_0.IsHomed THEN
					MpRoboArm6Axis_0.Home := FALSE;
					(*Step := ROBOTCTRL_READY;*)
					(*	Step_State := 'READY';*)
					MpPackMLStateComplete(gPackMLCore, 1);

				END_IF;

		END_CASE;

	END_IF;
END_ACTION
```

#### Starting.st
```iecst
ACTION Starting:

	IF MpPackMLStateIsActive(gPackMLCore,
		mpPACKML_STATE_STARTING,
		1) THEN

		MpPackMLMode_Auto.Start := 0;

		PackML_State := 'STARTING';

		Camera_0.ImageAcq := 0;

		DetectedSquares := 0;
		DetectedScrew := 0;
		DetectedScrewWasher := 0;
		DetectedWrench := 0;

		FOR i := 0 TO 13 DO
			//SQUARES DETECTION
			gSquareArray[Camera_0.ModelNumArray[i]-1] := Camera_0.PixelCntSquareArray[i] < PixelRange_0.HolderLimit;
			gIsPosGood[Camera_0.ModelNumArray[i]-1] := Camera_0.PixelCntSquareArray[i] < PixelRange_0.HolderLimit;
			IF Camera_0.PixelCntSquareArray[i] < PixelRange_0.HolderLimit THEN
				DetectedSquares := DetectedSquares + 1;
			END_IF

			IF Camera_0.PixelCntSquareArray[i] < 50 THEN
				//NOTHING
				gActPos[Camera_0.ModelNumArray[i]-1] := 0;
				gElementsArray[Camera_0.ModelNumArray[i]-1] := 0;
				DetectedScrew := 0;
				DetectedScrewWasher := 0;
				DetectedWrench := 0;
			ELSIF Camera_0.PixelCntSquareArray[i] < PixelRange_0.ScrewLimit THEN
				//SCREW
				gActPos[Camera_0.ModelNumArray[i]-1] := 1;
				gElementsArray[Camera_0.ModelNumArray[i]-1] := 1;
				DetectedScrew := DetectedScrew + 1;
			ELSIF Camera_0.PixelCntSquareArray[i] < PixelRange_0.WasherBoltLimit THEN
				//WASHER BOLT
				gActPos[Camera_0.ModelNumArray[i]-1] := 2;
				gElementsArray[Camera_0.ModelNumArray[i]-1] := 2;
				DetectedScrewWasher := DetectedScrewWasher + 1;
			ELSIF Camera_0.PixelCntSquareArray[i] < PixelRange_0.WrenchLimit THEN
				//WRENCH
				gActPos[Camera_0.ModelNumArray[i]-1] := 4;
				gElementsArray[Camera_0.ModelNumArray[i]-1] := 4;
				DetectedWrench := DetectedWrench + 1;
			ELSE
				gActPos[Camera_0.ModelNumArray[i]-1] := 0;
				gElementsArray[Camera_0.ModelNumArray[i]-1] := 0;
				DetectedScrew := 0;
				DetectedScrewWasher := 0;
				DetectedWrench := 0;
			END_IF;

		END_FOR;

		CASE Step OF
			ROBOTCTRL_CHECK: 	//checking if aim targets are available

				AimIsGood:=TRUE;
				FOR x:=0  TO SizeOfArray DO
					IF gAimPos[x]>0 THEN
						IF (gIsPosGood[x]=FALSE) THEN
							Step:=ROBOTCTRL_ERROR_WRONG_AIM;
							Step_State := 'ERROR_WRONG_AIM';
							AimIsGood:=0;
						END_IF;
					END_IF;
				END_FOR;
				IF AimIsGood=TRUE THEN
					y:=0;
					P1P2_Ok:=0;
					Step:=ROBOTCTRL_CALCULATE;
					Step_State := 'CALCULATE';
					Camera_0.diTrigger := 0;
					MpPackMLStateComplete(gPackMLCore, 1);
				END_IF;

			ROBOTCTRL_ERROR_WRONG_AIM:
				//handling wrong target error
				doVisError:=TRUE;
				IF diAck THEN
					doVisError:=FALSE;

					Step:=ROBOTCTRL_CHECK;
					Step_State := 'CHECK';
				END_IF;

		END_CASE;

	END_IF
END_ACTION
```

#### Stopped.st
```iecst
ACTION Stopped:
	IF MpPackMLStateIsActive(gPackMLCore,
		mpPACKML_STATE_STOPPED,
		1) THEN

		PackML_State := 'STOPPED';
		MpRoboArm6Axis_0.Power := FALSE;

		IF diReset THEN
			Step := ROBOTCTRL_POWER;
			Step_State := 'POWER';
			MpPackMLMode_Auto.Reset := TRUE;
			diReset := FALSE;
		END_IF

	END_IF

END_ACTION
```

#### Stopping.st
```iecst
ACTION Stopping:
	IF MpPackMLStateIsActive(gPackMLCore,
		mpPACKML_STATE_STOPPING,
		1) THEN

		PackML_State := 'STOPPING';
		gCompliteFlag:=FALSE;
		//STOP EVERYTHING
		MpRoboArm6Axis_0.Stop := TRUE;
		IF NOT MpRoboArm6Axis_0.InMotion THEN
				MpRoboArm6Axis_0.Stop := FALSE;
			MpRoboArm6Axis_0.Power := FALSE;
			emptyPos:=0;
			diStop := 0;

		//	IF NOT MpRoboArm6Axis_0.InMotion AND (NOT MpRoboArm6Axis_0.PowerOn) THEN

				MpPackMLStateComplete(gPackMLCore, 1);
		//	END_IF;

	END_IF;

	END_IF

END_ACTION
```

#### Unhold.st
```iecst
ACTION Unhold:

	IF MpPackMLStateIsActive(gPackMLCore,
		mpPACKML_STATE_UNHOLDING,
		1) THEN

		PackML_State := 'UNHOLD';

		MpRoboArm6Axis_0.Continue := 1;
		MpPackMLMode_Auto.Unhold := 0;
		IF  MpRoboArm6Axis_0.InMotion THEN
			MpRoboArm6Axis_0.Continue:=0;
//			Step:=ROBOTCTRL_MOVE;
//			Step_State := 'MOVE';
			MpPackMLStateComplete(gPackMLCore, 1);
			MpPackMLMode_Auto.Hold := 0;
		END_IF
	END_IF

END_ACTION
```

### Program Logical/Robot/PackML/PackML_Logic

#### Main.st
```iecst
PROGRAM _INIT
	MpPackMLCore_0.MpLink := ADR(gPackMLCore);
	MpPackMLCore_0.Enable := TRUE;

	MpPackMLMode_Auto.MpLink := ADR(gPackMLCore);
	MpPackMLMode_Auto.Enable := TRUE;
	MpPackMLMode_Auto.ModeID := 1;

	MpPackMLMode_SemiAuto.MpLink := ADR(gPackMLCore);
	MpPackMLMode_SemiAuto.Enable := TRUE;
	MpPackMLMode_SemiAuto.ModeID := 2;

	MpPackMLMode_Manual.MpLink := ADR(gPackMLCore);
	MpPackMLMode_Manual.Enable := TRUE;
	MpPackMLMode_Manual.ModeID := 3;

	MpPackMLMode_Auto.Activate := 0;
	MpPackMLMode_SemiAuto.Activate := 0;
	MpPackMLMode_Manual.Activate := 0;

END_PROGRAM

PROGRAM _CYCLIC
	MpPackMLCore_0();
	MpPackMLMode_Auto();
	MpPackMLMode_SemiAuto();
	MpPackMLMode_Manual();

	MpPackMLMode_Auto.Activate := 0;
	MpPackMLMode_SemiAuto.Activate := 0;
	MpPackMLMode_Manual.Activate := 0;

	MpPackMLMode_Auto.Activate := diAuto AND (NOT diSemiAuto) AND (NOT diManual);
	MpPackMLMode_SemiAuto.Activate := diSemiAuto AND (NOT diAuto) AND (NOT diManual);
	MpPackMLMode_Manual.Activate := diManual AND (NOT diAuto) AND (NOT diSemiAuto);
END_PROGRAM

PROGRAM _EXIT
	MpPackMLCore_0.Enable := 0;
	MpPackMLMode_Auto.Enable := 0;
	MpPackMLMode_SemiAuto.Enable := 0;
	MpPackMLMode_Manual.Enable := 0;

	MpPackMLCore_0();
	MpPackMLMode_Auto();
	MpPackMLMode_SemiAuto();
	MpPackMLMode_Manual();

END_PROGRAM
```

### Program Logical/Robot/PackML/PackML_Manual

#### Completing.st
```iecst
ACTION Completing:

END_ACTION
```

#### Execute.st
```iecst
ACTION Execute:

END_ACTION
```

#### Main.st
```iecst
PROGRAM _INIT
	(* Insert code here *)
	Axis;

END_PROGRAM

PROGRAM _CYCLIC
	Starting;
	Idle;
	Stopping;
	Resetting;
	Execute;
	Completing;
	Complete;
	Stopped;

	VelocityQ;
	doMagnet;
	VelocityQQ;
	RoboParameters.Jog.Velocity[0] := VelocityQ1;
	RoboParameters.Jog.Velocity[1] := VelocityQ2;
	RoboParameters.Jog.Velocity[2] := VelocityQ3;
	RoboParameters.Jog.Velocity[3] := VelocityQ4;
	RoboParameters.Jog.Velocity[4] := VelocityQ5;
	RoboParameters.Jog.Velocity[5] := VelocityQ6;

	IF cartezianVSjog THEN
		RoboParameters.Jog.CoordSystem := 10;
	ELSE
		RoboParameters.Jog.CoordSystem := 0;
	END_IF

	IF diManual THEN
		RoboParameters.ProgramName := 'HOME.st';
	ELSE
		RoboParameters.ProgramName := 'Robotic.st';
	END_IF

END_PROGRAM

PROGRAM _EXIT
	(* Insert code here *)

END_PROGRAM
```

#### Starting.st
```iecst
ACTION Starting:

END_ACTION
```

### Program Logical/Robot/PackML/PackML_SemiAuto

#### Complete.st
```iecst
ACTION Complete:

END_ACTION
```

#### Main.st
```iecst
PROGRAM _INIT
	(* Insert code here *)
	 Axis;
END_PROGRAM

PROGRAM _CYCLIC
	Starting;
	Idle;
	Stopping;
	Resetting;
	Execute;
	Completing;
	Complete;
	Stopped;

END_PROGRAM

PROGRAM _EXIT
	(* Insert code here *)

END_PROGRAM
```

#### Stopped.st
```iecst
ACTION Stopped:

END_ACTION
```

#### Stopping.st
```iecst
ACTION Stopping:

END_ACTION
```

### HOME.st
```iecst
VAR

	A : McAxisTargetType := (JointAxis:=[0, 0, -90, 0, 90, 0], SlaveAxis:=[100]);

END_VAR

	PROGRAM _MAIN

	Feedrate(10000);    //move with reduced speed
	MoveA(A); //move HOME
	END_PROGRAM
```

### Robotic.st
```iecst
VAR {AT PLC}
P2up : McPointType;
P2 : McPointType;
P1up : McPointType;
P1 : McPointType;
P0 : McPointType;
HOME : McPointType;
PZ : McPointType;
A : McAxisTargetType;
doMagnet : BOOL;
y : USINT;
gWait : REAL;
MaxSpeed : DINT;
LowSpeed : DINT;

END_VAR

	PROGRAM _MAIN

	Feedrate(MaxSpeed);    //move with reduced speed

	IF y=0 THEN
		MoveA(A); //move HOME
	END_IF;

//	MoveJ(P0);   //move to lower HOME pose

	MoveL(P1up); //move over the aim 1 pose
	Feedrate(LowSpeed);

	MoveL(P1);  //move to aim 1

	DO_PATH_SYNCH
	doMagnet := TRUE;
	END_PATH_SYNCH

	WaitTime(gWait);
	MoveL(P1up); //move over the aim 1 pose
	Feedrate(MaxSpeed);
	MoveL(P2up); //move over the aim 2 pose
	Feedrate(LowSpeed);

	MoveL(P2);    //move to aim 2
	DO_PATH_SYNCH
	doMagnet := FALSE;
	END_PATH_SYNCH
	WaitTime(gWait);

	MoveL(P2up); //move over the aim 2 pose
	Feedrate(MaxSpeed);

	//	MoveL(P0);   //move to lower HOME pose
	IF y=2 THEN
		MoveJ(HOME); //move to  HOME
	END_IF;

END_PROGRAM
```

### Program Logical/Services/File_explorer (IEC)

#### Types.typ
```iecst
TYPE
	TabInfo : 	STRUCT
		LastModified : ARRAY[0..49]OF DATE_AND_TIME;
		Type : ARRAY[0..49]OF MpFileManagerUIItemTypeEnum;
		Size : ARRAY[0..49]OF UDINT;
		Name : ARRAY[0..49]OF STRING[80];
		SelectedRow : USINT;
		NumberOfElements : INT;
	END_STRUCT;
END_TYPE
```

#### Main.st
```iecst
PROGRAM _INIT
	(* Insert code here *)
	MpFileMngSetup.FileListSize := 50;
	MpFileManagerUI_0(MpLink := ADR(gFileManagerUI), Enable :=1 , ErrorReset :=0 , UISetup :=MpFileMngSetup , UIConnect :=ADR(MpFileMngConnect));
	MpFileMngConnect.DeviceList.DeviceNames[0] := 'FilesDir';
	sortOrder[0] := '{"value":"0", "text":"Alphabetic (ascending)"}';
	sortOrder[1] := '{"value":"1", "text":"Alphabetic (descending)"}';
	sortOrder[2] := '{"value":"2", "text":"By size (ascending)"}';
	sortOrder[3] := '{"value":"3", "text":"By size (descending)"}';
	sortOrder[4] := '{"value":"4", "text":"By date (ascending))"}';
	sortOrder[5] := '{"value":"5", "text":"By date (descending)"}';
END_PROGRAM

PROGRAM _CYCLIC
	(* Insert code here *)
	MpFileManagerUI_0();
	tabInfo.NumberOfElements := 0;

	CASE chosenSortOrder OF
		0:
			MpFileMngConnect.File.SortOrder := mpFILE_SORT_BY_NAME_ASC;
		1:
			MpFileMngConnect.File.SortOrder := mpFILE_SORT_BY_NAME_DESC;
		2:
			MpFileMngConnect.File.SortOrder := mpFILE_SORT_BY_SIZE_ASC;
		3:
			MpFileMngConnect.File.SortOrder := mpFILE_SORT_BY_SIZE_DES;
		4:
			MpFileMngConnect.File.SortOrder := mpFILE_SORT_BY_MOD_TIME_ASC;
		5:
			MpFileMngConnect.File.SortOrder := mpFILE_SORT_BY_MOD_TIME_DESC;
	END_CASE

	IF MpFileMngConnect.MessageBox.Type = mpFILE_MSG_OK THEN
		messageType := 'OK';
	ELSIF MpFileMngConnect.MessageBox.Type = mpFILE_MSG_CONFIRM_DELETE THEN
		messageType := 'DELETE';
	ELSIF MpFileMngConnect.MessageBox.Type = mpFILE_MSG_CONFIRM_OVERWRITE THEN
		messageType := 'OVERWRITE';
	ELSIF MpFileMngConnect.MessageBox.Type = mpFILE_MSG_BUSY THEN
		messageType := 'BUSY';
	END_IF

	FOR iFile := 0 TO 49 BY 1 DO
		(* create arrays with file properties *)
//		IF tabInfo.NumberOfElements >= iFile THEN
			brsmemcpy(ADR(tabInfo.Name[iFile]), ADR(MpFileMngConnect.File.List.Items[iFile].Name), SIZEOF(tabInfo.Name[iFile]));
			brsmemcpy(ADR(tabInfo.Size[iFile]), ADR(MpFileMngConnect.File.List.Items[iFile].Size), SIZEOF(tabInfo.Size[iFile]));
			brsmemcpy(ADR(tabInfo.Type[iFile]), ADR(MpFileMngConnect.File.List.Items[iFile].ItemType), SIZEOF(tabInfo.Type[iFile]));
			brsmemcpy(ADR(tabInfo.LastModified[iFile]), ADR(MpFileMngConnect.File.List.Items[iFile].LastModified), SIZEOF(tabInfo.LastModified[iFile]));
//		END_IF

		IF tabInfo.SelectedRow = iFile THEN
			MpFileMngConnect.File.List.Items[iFile].IsSelected := TRUE;
		END_IF
		(* numbers of elements in the table *)
		IF tabInfo.Type[iFile] <> mpFILE_ITEM_TYPE_NONE THEN
			//			tabInfo.NumberOfElements := iFile;
			tabInfo.NumberOfElements := tabInfo.NumberOfElements + 1;
		END_IF

		CASE tabInfo.Type[iFile] OF
			mpFILE_ITEM_TYPE_FOLDER:
				itemType[iFile] := 'Folder';
			mpFILE_ITEM_TYPE_FILE:
				itemType[iFile] := 'Plik';
			mpFILE_ITEM_TYPE_TXT:
				itemType[iFile] := 'Plik tekstowy';
			mpFILE_ITEM_TYPE_HTML:
				itemType[iFile] := 'Plik HTML';
			mpFILE_ITEM_TYPE_XLS:
				itemType[iFile] := 'Plik XLS';
			mpFILE_ITEM_TYPE_XML:
				itemType[iFile] := 'Plik XML';
			mpFILE_ITEM_TYPE_CSV:
				itemType[iFile] := 'Plik CSV';
			mpFILE_ITEM_TYPE_JPG:
				itemType[iFile] := 'Plik JPG';
			mpFILE_ITEM_TYPE_BMP:
				itemType[iFile] := 'Plik BMP';
			mpFILE_ITEM_TYPE_UNKNOWN:
				itemType[iFile] := 'Plik nieznany';
			END_CASE
	END_FOR

	tableShowLimit := tabInfo.NumberOfElements - 1;
	tableConfig := '{"specRows": [ {"from":0, "to":';
	brsitoa(tableShowLimit,ADR(tempString));
	brsstrcat(ADR(tableConfig),ADR(tempString));
	brsstrcat(ADR(tableConfig),ADR(', "visible":true}, {"from":'));
	brsitoa(tabInfo.NumberOfElements,ADR(tempString));
	brsstrcat(ADR(tableConfig),ADR(tempString));
	brsstrcat(ADR(tableConfig),ADR(', "to":49, "visible":false}]}'));

//		TableConfig := '{"specRows": [ ';
//		FOR Index:=0 TO MAX_ORDERS_NUM_MINUS_ONE DO
//			IF Index <> 0 THEN
//				brsstrcat(ADR(TableConfig), ADR(','));
//			END_IF;
//			brsstrcat(ADR(TableConfig), ADR('{"index":'));
//			brsitoa(Index, ADR(IndexStr)); (*write int_value to the string*)
//			brsstrcat(ADR(TableConfig), ADR(IndexStr));
//
//			//    IF  (OrderLengths[Index] = 0) AND (OrderCounts[Index] = 0) THEN
//			IF  (OrderLengths[Index] = 0) THEN
//
//				brsstrcat(ADR(TableConfig), ADR(', "visible":false}'));
//			ELSE
//				brsstrcat(ADR(TableConfig), ADR(', "visible":true}'));
//			END_IF;
//
//			IF (Index = MAX_ORDERS_NUM_MINUS_ONE) THEN
//				brsstrcat(ADR(TableConfig), ADR(']}'));
//			END_IF;
//		END_FOR;
//		(* Return true *)
//		CreateTableConfig := TRUE;

END_PROGRAM

PROGRAM _EXIT
	(* Insert code here *)
	MpFileManagerUI_0.Enable := FALSE;
	MpFileManagerUI_0();
END_PROGRAM
```

### Program Logical/Services/AuditPckg/AuditProgram (IEC)

#### Variables.var
```iecst
VAR
	MpAuditTrail_0 : MpAuditTrail := (0);
	TriggerEvent : BOOL := FALSE;
	TypeVar : WSTRING[100] := "0";
	MessageVar : WSTRING[100] := "0";
	CommentVar : WSTRING[100] := "0";
	Status : DINT := 0;
END_VAR
```

#### Cyclic.ld
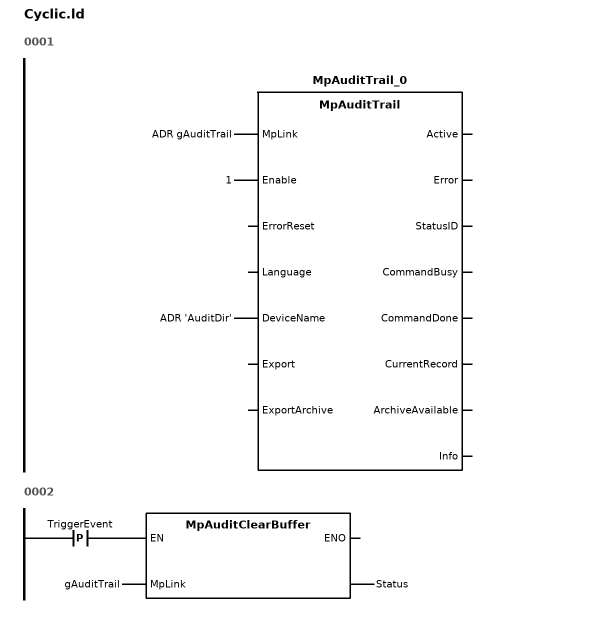
Ladder, written as Structured Text:
```iecst
PROGRAM _CYCLIC
VAR
    _e1 : R_TRIG;
END_VAR
(* Network 1 *)
MpAuditTrail_0(MpLink := ADR(gAuditTrail), Enable := 1, DeviceName := ADR('AuditDir'));

(* Network 2 *)
_e1(CLK := TriggerEvent);
IF _e1.Q THEN Status := MpAuditClearBuffer(MpLink := gAuditTrail); END_IF;
END_PROGRAM
```

### Program Logical/Services/AlarmClearHistory (IEC)

#### Variables.var
```iecst
VAR
	ClearHistory : BOOL;
	ClearHistoryOutput : DINT;
	ClearHistoryStatus : BOOL;
END_VAR
```

#### Cyclic.ld
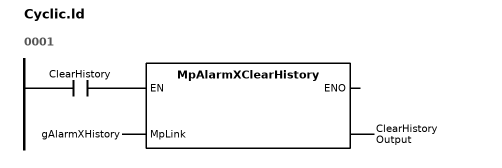
Ladder, written as Structured Text:
```iecst
PROGRAM _CYCLIC
(* Network 1 *)
IF ClearHistory THEN ClearHistoryOutput := MpAlarmXClearHistory(MpLink := gAlarmXHistory); END_IF;
END_PROGRAM
```

### Program Logical/Services/OpcCtrl (IEC)

#### Types.typ
```iecst
TYPE
	Safety_type : 	STRUCT  (*Struktura Safety. Logika: 0 - E-Stop wcisniety / Klatka otwarta*)
		EStop : BOOL; (*Stan Safety: E-Stop na klatce*)
		EStopPanel : BOOL; (*Stan Safety:  E-Stop na panelu*)
		GuardingDoor : BOOL; (*Stan Safety:  Drzwi klatki*)
		diEStop : BOOL; (*Stan wejscia: E-Stop na klatce*)
		diEStopPanel : BOOL; (*Stan wejscia: E-Stop na panelu*)
		diGuardDoor1 : BOOL; (*Stan wejscia: Drzwi klatki - kanal 1*)
		diGuardDoor2 : BOOL; (*Stan wejscia: Drzwi klatki - kanal 2*)
		SafeChannelOK1 : BOOL; (*Stan poprawnego dzialania SO1*)
		SafeChannelOK2 : BOOL; (*Stan poprawnego dzialania SO2*)
		doAcoposEnable1 : BOOL; (*Stan wyjsc Safety (Enable Acoposa 1)*)
		doAcoposEnable2 : BOOL; (*Stan wyjsc Safety (Enable Acoposa 2)*)
	END_STRUCT;
END_TYPE
```

#### Variables.var
```iecst
(*--- Obsluga odczytu danych z serwera OPC UA ---*)
(*   Laczenie z serwerem*)
VAR
	UA_Connect_0 : UA_Connect; (*Struktura do laczenia z serwerem*)
	ExecuteConnect_0 : BOOL; (*Wykonanie proby polaczenia z serwerem*)
	SessionConnectInfo_0 : UASessionConnectInfo; (*Informacje o sesji (protokol, dane logowanie, zabezpiczenia)*)
	ConnectionHdl : DWORD := 0;
	ErrorID : DWORD; (*ID bledu (pobierane z wszystkich blokow)*)
END_VAR
(*   Pobieranie indeksu przestrzeni nazw*)
VAR
	UA_GetNamespaceIndex_0 : UA_GetNamespaceIndex;
	ExecuteGetnamespaceindex_0 : BOOL;
	NamespaceIndex : UINT := 0;
END_VAR
(*   Uchyt do danego noda*)
VAR
	UA_NodeGetHandleList_0 : UA_NodeGetHandleList;
	ExecuteNodeGetHandleList_0 : BOOL;
	NodeIDs_0 : ARRAY[0..MAX_INDEX_NODELIST] OF UANodeID; (*Dane o zmiennych, ktore pobieramy z serwera*)
	NodeHdls : ARRAY[0..MAX_INDEX_NODELIST] OF DWORD;
END_VAR
(*   Odczyt danych*)
VAR
	UA_ReadList_0 : UA_ReadList;
	ExecuteReadList_0 : BOOL;
	NodeAddInfo_0 : ARRAY[0..MAX_INDEX_NODELIST] OF UANodeAdditionalInfo;
	Variables_Rd0 : ARRAY[0..MAX_INDEX_NODELIST] OF STRING[255]; (*Dane o zmiennych, do ktorych zapisujemy dane z serwera*)
END_VAR
(*   Zapis danych (nie jest uzywany)*)
VAR
	UA_WriteList_0 : UA_WriteList;
	ExecuteWriteList_0 : BOOL;
	Variables_Wr0 : ARRAY[0..MAX_INDEX_NODELIST] OF STRING[255];
END_VAR
(*   Zwolnienie uchytu danego noda*)
VAR
	UA_NodeReleaseHandleList_0 : UA_NodeReleaseHandleList;
	ExecuteNodeReleaseHandleList_0 : BOOL;
END_VAR
(*   Rozlaczenie z serwerem*)
VAR
	UA_Disconnect_0 : UA_Disconnect;
	ExecuteDisconnect_0 : BOOL;
END_VAR
(*--- Maszyna stanow ---*)
VAR
	ActState : USINT; (*Aktualny stan*)
END_VAR
VAR CONSTANT
	STATE_IDLE : USINT := 0; (*Stan wywolania proby polaczenia*)
	STATE_CONNECT : USINT := 1; (*Polaczenie z serwerem*)
	STATE_GET_NAMESPACE : USINT := 2; (*Pobranie przestrzeni nazw*)
	STATE_GET_HANDLE : USINT := 3; (*Przygotowanie uchytu*)
	STATE_READY_TO_READ : USINT := 10; (*Gotowosc do odczytu*)
	STATE_READ : USINT := 11; (*Realizacja odczytu danych*)
	STATE_RELEASE_HANDLE : USINT := 20; (*Zwolnienie uchytu*)
	STATE_DISCONNECT : USINT := 21; (*Rozlaczenie polaczenia z serwerem*)
	STATE_ERROR : USINT := 100; (*Stan obslugi bledow*)
	STATE_BACK_FROM_ERROR : USINT := 101; (*Stan powrotu ze stanu bledu*)
END_VAR
(*--- Struktura Safety ---*)
VAR
	SafetyLocal : Safety_type; (*Struktura przechowujaca informacje o stanie modulow Safety*)
END_VAR
(*--- Temporary ---*)
VAR
	Escape : BOOL; (*Zmienna tymczasowa wykorzystywana do debugowania programu*)
	LeaveIdel : BOOL; (*Zmienna tymczasowa wykorzystywana do debugowania programu*)
	MoveRead : BOOL; (*Zmienna tymczasowa wykorzystywana do debugowania programu*)
END_VAR
```

#### Main.st
```iecst
PROGRAM _INIT

	// Deklaracja podstawowych parametrow sesji klienta OPC UA
	SessionConnectInfo_0.SecurityMsgMode := UASecurityMsgMode_None;
	SessionConnectInfo_0.SecurityPolicy := UASecurityPolicy_None;
	SessionConnectInfo_0.TransportProfile := UATP_UATcp;
	SessionConnectInfo_0.UserIdentityToken.UserIdentityTokenType := UAUITT_Username;
	SessionConnectInfo_0.UserIdentityToken.TokenParam1 := 'admin';
	SessionConnectInfo_0.UserIdentityToken.TokenParam2 := 'password';
	SessionConnectInfo_0.SessionTimeout := T#1m;
	SessionConnectInfo_0.MonitorConnection := T#10s;

END_PROGRAM

PROGRAM _CYCLIC

	// Wywolanie funkcji polaczenia z serwerem
	UA_Connect_0(Execute := ExecuteConnect_0,
		ServerEndpointUrl := 'opc.tcp://192.168.0.115:4841',
	SessionConnectInfo := SessionConnectInfo_0,
	Timeout := T#10s);

//	UA_Connect_0(Execute := ExecuteConnect_0,
//		ServerEndpointUrl := 'opc.tcp://192.168.0.150:4841',
//	SessionConnectInfo := SessionConnectInfo_0,
//	Timeout := T#10s);

	// Wywolanie funkcji pobrania Namespace serwera
	UA_GetNamespaceIndex_0(Execute := ExecuteGetnamespaceindex_0,
		ConnectionHdl := ConnectionHdl,
		NamespaceUri := 'urn:B&R/pv/',
	Timeout := T#5s);

	// Wywolanie funkcji tworzacej uchtywy do zmiennych
	UA_NodeGetHandleList_0(Execute := ExecuteNodeGetHandleList_0,
		ConnectionHdl := ConnectionHdl,
		NodeIDCount := 11,
		NodeIDs := NodeIDs_0,
		Timeout := T#10s);

	// Odczyt poszczegolnych stanow zmiennych z serwera (sterownika safety)
	UA_ReadList_0(Execute := ExecuteReadList_0,
		ConnectionHdl := ConnectionHdl,
		NodeHdlCount := 11,
		NodeHdls := NodeHdls,
		NodeAddInfo := NodeAddInfo_0,
		Timeout := T#10s,
	Variables := Variables_Rd0);

	// Implementacja funkcjonalnosci zwolnienia uchyty - nie wykorzystywana, lecz mozliwa do wywolania
	UA_NodeReleaseHandleList_0(Execute := ExecuteNodeReleaseHandleList_0,
		ConnectionHdl := ConnectionHdl,
		NodeHdlCount := 11,
		NodeHdls := NodeHdls,
		Timeout := T#10s);

	// Implementacja funkcjonalnosci rozlaczenia polaczenia z serwerem - nie wykorzystywana, lecz mozliwa do wywolania
	UA_Disconnect_0(Execute := ExecuteDisconnect_0,
		ConnectionHdl := ConnectionHdl,
		Timeout := T#10s);

	CASE ActState OF
		STATE_IDLE:

				// Rozpoczecie wykonywania sekwencji odczytu danych
				ActState := STATE_CONNECT;
				ExecuteConnect_0 := TRUE;

		STATE_CONNECT:

			// UA_Connect - realizuje polaczenie z serwerem OPC UA
			IF (UA_Connect_0.Busy = 0) THEN
				ExecuteConnect_0 := 0;
				IF (UA_Connect_0.Done = 1) THEN								// Operacja wykonana poprawnie - wywolanie i przejscie do kolejnego kroku
					ErrorID := 0;
					ConnectionHdl := UA_Connect_0.ConnectionHdl;
					ExecuteGetnamespaceindex_0 := TRUE;
					ActState := STATE_GET_NAMESPACE;
				END_IF
				IF (UA_Connect_0.Error = 1) THEN							// Operacja nieudana (blad) - obsluga bledow
					ErrorID := UA_Connect_0.ErrorID;
					ConnectionHdl := 0;
					ActState := STATE_ERROR;
				END_IF
			END_IF

		STATE_GET_NAMESPACE:

			// UA_GetNamespaceIndex - odczytanie indeksow poszczegolnych przestrzeni nazw serwera
			IF (UA_GetNamespaceIndex_0.Busy = 0) THEN
				ExecuteGetnamespaceindex_0 := 0;
				IF (UA_GetNamespaceIndex_0.Done = 1) THEN
					ErrorID:= 0;
					NamespaceIndex := UA_GetNamespaceIndex_0.NamespaceIndex;
					ExecuteNodeGetHandleList_0 := TRUE;

					// Przypisanie poszczegolnych przestrzeni nazw z serwera odpowiednim indeksa
					NodeIDs_0[0].NamespaceIndex := NamespaceIndex;
					NodeIDs_0[0].Identifier := '::SafetyProg:EStop';
					NodeIDs_0[0].IdentifierType := UAIdentifierType_String;

					NodeIDs_0[1].NamespaceIndex := NamespaceIndex;
					NodeIDs_0[1].Identifier := '::SafetyProg:EStopPanel';
					NodeIDs_0[1].IdentifierType := UAIdentifierType_String;

					NodeIDs_0[2].NamespaceIndex := NamespaceIndex;
					NodeIDs_0[2].Identifier := '::SafetyProg:GuardDoor';
					NodeIDs_0[2].IdentifierType := UAIdentifierType_String;

					NodeIDs_0[3].NamespaceIndex := NamespaceIndex;
					NodeIDs_0[3].Identifier := '::SafetyProg:diEStop';
					NodeIDs_0[3].IdentifierType := UAIdentifierType_String;

					NodeIDs_0[4].NamespaceIndex := NamespaceIndex;
					NodeIDs_0[4].Identifier := '::SafetyProg:diEStopPanel';
					NodeIDs_0[4].IdentifierType := UAIdentifierType_String;

					NodeIDs_0[5].NamespaceIndex := NamespaceIndex;
					NodeIDs_0[5].Identifier := '::SafetyProg:diGuardDoor1';
					NodeIDs_0[5].IdentifierType := UAIdentifierType_String;

					NodeIDs_0[6].NamespaceIndex := NamespaceIndex;
					NodeIDs_0[6].Identifier := '::SafetyProg:diGuardDoor2';
					NodeIDs_0[6].IdentifierType := UAIdentifierType_String;

					NodeIDs_0[7].NamespaceIndex := NamespaceIndex;
					NodeIDs_0[7].Identifier := '::SafetyProg:SafeOutputOk1';
					NodeIDs_0[7].IdentifierType := UAIdentifierType_String;

					NodeIDs_0[8].NamespaceIndex := NamespaceIndex;
					NodeIDs_0[8].Identifier := '::SafetyProg:SafeOutputOk2';
					NodeIDs_0[8].IdentifierType := UAIdentifierType_String;

					NodeIDs_0[9].NamespaceIndex := NamespaceIndex;
					NodeIDs_0[9].Identifier := '::SafetyProg:gdoAcoposEnable1';
					NodeIDs_0[9].IdentifierType := UAIdentifierType_String;

					NodeIDs_0[10].NamespaceIndex := NamespaceIndex;
					NodeIDs_0[10].Identifier := '::SafetyProg:gdoAcoposEnable2';
					NodeIDs_0[10].IdentifierType := UAIdentifierType_String;

					ActState := STATE_GET_HANDLE;

				END_IF
				IF (UA_GetNamespaceIndex_0.Error = 1) THEN
					ErrorID:= UA_GetNamespaceIndex_0.ErrorID;
					NamespaceIndex := 0;
					ActState := STATE_ERROR;
				END_IF
			END_IF

		STATE_GET_HANDLE:

			// UA_NodeGetHandle - uchyt do noda
			IF (UA_NodeGetHandleList_0.Busy = 0) THEN
				ExecuteNodeGetHandleList_0 := 0;
				IF (UA_NodeGetHandleList_0.Done = 1) THEN
					ErrorID:= 0;
					NodeHdls := UA_NodeGetHandleList_0.NodeHdls;
					ExecuteReadList_0 := TRUE;
					ActState := STATE_READY_TO_READ;
				END_IF
				IF (UA_NodeGetHandleList_0.Error = 1) THEN
					ErrorID:= UA_NodeGetHandleList_0.ErrorID;
					NodeHdls[0] := 0;
					NodeHdls[1] := 0;
					NodeHdls[2] := 0;
					NodeHdls[3] := 0;
					NodeHdls[4] := 0;
					NodeHdls[5] := 0;
					NodeHdls[6] := 0;
					NodeHdls[7] := 0;
					NodeHdls[8] := 0;
					NodeHdls[9] := 0;
					NodeHdls[10] := 0;
					ActState := STATE_ERROR;
				END_IF
			END_IF

		STATE_READY_TO_READ:

			NodeAddInfo_0[0].AttributeId := UAAI_Value;
			NodeAddInfo_0[0].IndexRangeCount := 0;

			NodeAddInfo_0[1].AttributeId := UAAI_Value;
			NodeAddInfo_0[1].IndexRangeCount := 0;

			NodeAddInfo_0[2].AttributeId := UAAI_Value;
			NodeAddInfo_0[2].IndexRangeCount := 0;

			NodeAddInfo_0[3].AttributeId := UAAI_Value;
			NodeAddInfo_0[3].IndexRangeCount := 0;

			NodeAddInfo_0[4].AttributeId := UAAI_Value;
			NodeAddInfo_0[4].IndexRangeCount := 0;

			NodeAddInfo_0[5].AttributeId := UAAI_Value;
			NodeAddInfo_0[5].IndexRangeCount := 0;

			NodeAddInfo_0[6].AttributeId := UAAI_Value;
			NodeAddInfo_0[6].IndexRangeCount := 0;

			NodeAddInfo_0[7].AttributeId := UAAI_Value;
			NodeAddInfo_0[7].IndexRangeCount := 0;

			NodeAddInfo_0[8].AttributeId := UAAI_Value;
			NodeAddInfo_0[8].IndexRangeCount := 0;

			NodeAddInfo_0[9].AttributeId := UAAI_Value;
			NodeAddInfo_0[9].IndexRangeCount := 0;

			NodeAddInfo_0[10].AttributeId := UAAI_Value;
			NodeAddInfo_0[10].IndexRangeCount := 0;

			// Przypisanie przestrzeni nazw, do ktorych zmienna maja byc zapisywane
			Variables_Rd0[0] := '::OpcCtrl:SafetyLocal.EStop';
			Variables_Rd0[1] := '::OpcCtrl:SafetyLocal.EStopPanel';
			Variables_Rd0[2] := '::OpcCtrl:SafetyLocal.GuardingDoor';
			Variables_Rd0[3] := '::OpcCtrl:SafetyLocal.diEStop';
			Variables_Rd0[4] := '::OpcCtrl:SafetyLocal.diEStopPanel';
			Variables_Rd0[5] := '::OpcCtrl:SafetyLocal.diGuardDoor1';
			Variables_Rd0[6] := '::OpcCtrl:SafetyLocal.diGuardDoor2';
			Variables_Rd0[7] := '::OpcCtrl:SafetyLocal.SafeChannelOK1';
			Variables_Rd0[8] := '::OpcCtrl:SafetyLocal.SafeChannelOK2';
			Variables_Rd0[9] := '::OpcCtrl:SafetyLocal.doAcoposEnable1';
			Variables_Rd0[10] := '::OpcCtrl:SafetyLocal.doAcoposEnable1';

			ActState := STATE_READ;
			ExecuteReadList_0 := TRUE;

		STATE_READ:

			// UA_Read - odczyt danych
			IF (UA_ReadList_0.Busy = 0) THEN
				ExecuteReadList_0 := 0;
				IF (UA_ReadList_0.Done = 1) THEN
					ErrorID:= 0;
					ActState := STATE_READY_TO_READ;
				END_IF
				IF (UA_ReadList_0.Error = 1) THEN
					ErrorID:= UA_ReadList_0.ErrorID;
					SafetyLocal.EStop := FALSE;
					SafetyLocal.EStopPanel := FALSE;
					SafetyLocal.GuardingDoor := FALSE;
					SafetyLocal.diEStop := FALSE;
					SafetyLocal.diEStopPanel := FALSE;
					SafetyLocal.diGuardDoor1 := FALSE;
					SafetyLocal.diGuardDoor2 := FALSE;
					SafetyLocal.SafeChannelOK1 := FALSE;
					SafetyLocal.SafeChannelOK2 := FALSE;
					SafetyLocal.doAcoposEnable1 := FALSE;
					SafetyLocal.doAcoposEnable2 := FALSE;
					ActState := STATE_ERROR;
				END_IF
			END_IF

		STATE_RELEASE_HANDLE:

			(* UA_NodeReleaseHandle - release the handle for the node *)

			IF (UA_NodeReleaseHandleList_0.Busy = 0) THEN
				ExecuteNodeReleaseHandleList_0 := 0;
				IF (UA_NodeReleaseHandleList_0.Done = 1) THEN
					ErrorID:= 0;
					NodeHdls[0] := 0;
					NodeHdls[1] := 0;
					NodeHdls[2] := 0;
					NodeHdls[3] := 0;
					NodeHdls[4] := 0;
					NodeHdls[5] := 0;
					NodeHdls[6] := 0;
					NodeHdls[7] := 0;
					NodeHdls[8] := 0;
					NodeHdls[9] := 0;
					NodeHdls[10] := 0;
				END_IF
				IF (UA_NodeReleaseHandleList_0.Error = 1) THEN
					ErrorID:= UA_NodeReleaseHandleList_0.ErrorID;
				END_IF
			END_IF

		STATE_DISCONNECT:

			(* UA_Disconnect - disconnect from OPC UA Server *)

			IF (UA_Disconnect_0.Busy = 0) THEN
				ExecuteDisconnect_0 := 0;
				IF (UA_Disconnect_0.Done = 1) THEN
					ErrorID:= 0;
					ConnectionHdl := 0;
				END_IF
				IF (UA_Disconnect_0.Error = 1) THEN
					ErrorID:= UA_Disconnect_0.ErrorID;
				END_IF
			END_IF

		STATE_ERROR:

			// Aktywowanie alarmu o bledzie w komunikacji
			gSafety.CommunicationError := TRUE;

			// proba potwierdzenia alarmu
			IF gSafety.ComErrorAck THEN
				gSafety.ComErrorAck := FALSE;
				// Execute = FALSE pozwala na zresetowanie bledow
				ExecuteConnect_0 := FALSE;
				ExecuteGetnamespaceindex_0 := FALSE;
				ExecuteNodeGetHandleList_0 := FALSE;
				ExecuteReadList_0 := FALSE;
				ActState := STATE_BACK_FROM_ERROR;
			END_IF

		STATE_BACK_FROM_ERROR:

			// Powrot do proby laczenia z serwerem w przypadku, gdy bledy zostaly zresetowane
			IF (NOT UA_Connect_0.Error) AND NOT UA_GetNamespaceIndex_0.Error AND NOT UA_NodeGetHandleList_0.Error AND NOT UA_ReadList_0.Error THEN
//			IF Escape THEN
				ActState := STATE_IDLE;
			END_IF;

	END_CASE;

	// Zresetowanie alarmu o bledzie w komunikacji
	IF ErrorID = 0 THEN
		gSafety.CommunicationError := FALSE;
	END_IF;

	// Przypisanie odpowiednich zmiennych lokalnych do globalej struktury wykorzystywanej do kontroli Safety
	gSafety.diEStop := SafetyLocal.diEStop;
	gSafety.diEStopPanel := SafetyLocal.diEStopPanel;
	gSafety.diGuardDoor1 := SafetyLocal.diGuardDoor1;
	gSafety.diGuardDoor2 := SafetyLocal.diGuardDoor2;
	gSafety.EStop := SafetyLocal.EStop;
	gSafety.EStopPanel := SafetyLocal.EStopPanel;
	gSafety.GuardingDoor := SafetyLocal.GuardingDoor;
	gSafety.SafeChannelOK1 := SafetyLocal.SafeChannelOK1;
	gSafety.SafeChannelOK2 := SafetyLocal.SafeChannelOK2;
	gSafety.doAcoposEnable1 := SafetyLocal.doAcoposEnable1;
	gSafety.doAcoposEnable2 := SafetyLocal.doAcoposEnable2;

END_PROGRAM

PROGRAM _EXIT

END_PROGRAM
```

### Program Logical/Services/Alarms (IEC)

#### Main.st
```iecst
PROGRAM _INIT
	MpAlarmXCore_0.MpLink := ADR(gAlarmXCore0);
	MpAlarmXCore_0.Enable := TRUE;
	MpAlarmXHistory_0.MpLink := ADR(gAlarmXHistory);
	MpAlarmXHistory_0.Enable := TRUE;
END_PROGRAM

PROGRAM _CYCLIC
	MpAlarmXCore_0();
	MpAlarmXHistory_0();
END_PROGRAM

PROGRAM _EXIT
	MpAlarmXCore_0.Enable := FALSE;
	MpAlarmXHistory_0.Enable := FALSE;
	MpAlarmXCore_0();
	MpAlarmXHistory_0();
END_PROGRAM
```

### Program Logical/Camera/Elements_detection (IEC)

#### Main.st
```iecst
PROGRAM _INIT
	//CAMERA INITIAL VALUES
	Camera_0.Focus := 30000;
	Camera_0.ExposureTime := 40000;
	Camera_0.NumSearch := 14;
	Camera_0.Enable := 1;

	PixelRange_0.ScrewLimit := 200;
	PixelRange_0.WasherBoltLimit := 500;
	PixelRange_0.WrenchLimit := 2000;
	PixelRange_0.HolderLimit := 10000;

	///////////////////////////////
	DetectedSquares := 7;
	DetectedScrew := 1;
	DetectedScrewWasher := 1;
	DetectedWrench := 1;
	//////////////////////////////

END_PROGRAM

PROGRAM _CYCLIC
	//IMAGE ACQUISITION
	Camera_0.ImageAcq := Camera_0.diTrigger AND Camera_0.Ready;

	DetectedSquares := 0;
	DetectedScrew := 0;
	DetectedScrewWasher := 0;
	DetectedWrench := 0;

	FOR i := 0 TO 13 DO
		//SQUARES DETECTION
		gSquareArray[Camera_0.ModelNumArray[i]-1] := Camera_0.PixelCntSquareArray[i] < PixelRange_0.HolderLimit;
		gIsPosGood[Camera_0.ModelNumArray[i]-1] := Camera_0.PixelCntSquareArray[i] < PixelRange_0.HolderLimit;
		IF Camera_0.PixelCntSquareArray[i] < PixelRange_0.HolderLimit THEN
			DetectedSquares := DetectedSquares + 1;
		END_IF

		IF Camera_0.PixelCntSquareArray[i] < 50 THEN
			//NOTHING
			gActPos[Camera_0.ModelNumArray[i]-1] := 0;
			gElementsArray[Camera_0.ModelNumArray[i]-1] := 0;
		ELSIF Camera_0.PixelCntSquareArray[i] < PixelRange_0.ScrewLimit THEN
			//SCREW
			gActPos[Camera_0.ModelNumArray[i]-1] := 1;
			gElementsArray[Camera_0.ModelNumArray[i]-1] := 1;
			DetectedScrew := DetectedScrew + 1;
		ELSIF Camera_0.PixelCntSquareArray[i] < PixelRange_0.WasherBoltLimit THEN
			//WASHER BOLT
			gActPos[Camera_0.ModelNumArray[i]-1] := 2;
			gElementsArray[Camera_0.ModelNumArray[i]-1] := 2;
			DetectedScrewWasher := DetectedScrewWasher + 1;
		ELSIF Camera_0.PixelCntSquareArray[i] < PixelRange_0.WrenchLimit THEN
			//WRENCH
			gActPos[Camera_0.ModelNumArray[i]-1] := 4;
			gElementsArray[Camera_0.ModelNumArray[i]-1] := 4;
			DetectedWrench := DetectedWrench + 1;
		ELSE
			gActPos[Camera_0.ModelNumArray[i]-1] := 0;
			gElementsArray[Camera_0.ModelNumArray[i]-1] := 0;
		END_IF;

	END_FOR;

END_PROGRAM

PROGRAM _EXIT

END_PROGRAM
```

### Robotic.st - not listed in the package file held
```iecst
VAR {AT PLC}
P2up : McPointType;
P2 : McPointType;
P1up : McPointType;
P1 : McPointType;
P0 : McPointType;
HOME : McPointType;
PZ : McPointType;
A : McAxisTargetType;
doMagnet : BOOL;
y : USINT;
MaxSpeed : DINT;
LowSpeed : DINT;

END_VAR

	PROGRAM _MAIN

	Feedrate(MaxSpeed);    //move with reduced speed

	IF y=0 THEN
		MoveA(A); //move HOME
	END_IF;

//	MoveJ(P0);   //move to lower HOME pose

	MoveL(P1up); //move over the aim 1 pose
	Feedrate(LowSpeed);

	MoveL(P1);  //move to aim 1

	DO_PATH_SYNCH
	doMagnet := TRUE;
	END_PATH_SYNCH

	WaitTime(1);
	MoveL(P1up); //move over the aim 1 pose
	Feedrate(MaxSpeed);
	MoveL(P2up); //move over the aim 2 pose
	Feedrate(LowSpeed);

	MoveL(P2);    //move to aim 2
	DO_PATH_SYNCH
	doMagnet := FALSE;
	END_PATH_SYNCH
	WaitTime(1);

	MoveL(P2up); //move over the aim 2 pose
	Feedrate(MaxSpeed);

	//	MoveL(P0);   //move to lower HOME pose
	IF y=2 THEN
		MoveJ(HOME); //move to  HOME
	END_IF;

END_PROGRAM
```

### Variables.var
```iecst
VAR
	iFile : INT;
	MpFileManagerUI_0 : MpFileManagerUI;
	MpFileMngSetup : MpFileManagerUISetupType;
	MpFileMngConnect : MpFileManagerUIConnectType;
	tabInfo : TabInfo;
	messageType : STRING[80];
	tempString : STRING[200];
	tableConfig : STRING[200];
	testString : STRING[200] := '{"specRows": [ {"from":0, "to":3, "visible":true}, {"from":4, "to":49, "visible":false}]}';
	tableShowLimit : INT;
	sortOrder : ARRAY[0..5] OF STRING[80];
	chosenSortOrder : INT;
	itemType : ARRAY[0..49] OF STRING[80];
END_VAR
```

### Program Logical/PackML/PackML_Logic (IEC)

#### Main.st
```iecst
PROGRAM _INIT
	MpPackMLCore_0.MpLink := ADR(gPackMLCore);
	MpPackMLCore_0.Enable := TRUE;

	MpPackMLMode_Auto.MpLink := ADR(gPackMLCore);
	MpPackMLMode_Auto.Enable := TRUE;
	MpPackMLMode_Auto.ModeID := 1;

	MpPackMLMode_SemiAuto.MpLink := ADR(gPackMLCore);
	MpPackMLMode_SemiAuto.Enable := TRUE;
	MpPackMLMode_SemiAuto.ModeID := 2;

	MpPackMLMode_Manual.MpLink := ADR(gPackMLCore);
	MpPackMLMode_Manual.Enable := TRUE;
	MpPackMLMode_Manual.ModeID := 3;

	MpPackMLMode_Auto.Activate := 0;
	MpPackMLMode_SemiAuto.Activate := 0;
	MpPackMLMode_Manual.Activate := 0;

END_PROGRAM

PROGRAM _CYCLIC
	MpPackMLCore_0();
	MpPackMLMode_Auto();
	MpPackMLMode_SemiAuto();
	MpPackMLMode_Manual();

	MpPackMLMode_Auto.Activate := 0;
	MpPackMLMode_SemiAuto.Activate := 0;
	MpPackMLMode_Manual.Activate := 0;

	MpPackMLMode_Auto.Activate := diAuto AND (NOT diSemiAuto) AND (NOT diManual);
	MpPackMLMode_SemiAuto.Activate := diSemiAuto AND (NOT diAuto) AND (NOT diManual);
	MpPackMLMode_Manual.Activate := diManual AND (NOT diAuto) AND (NOT diSemiAuto);
END_PROGRAM

PROGRAM _EXIT
	MpPackMLCore_0.Enable := 0;
	MpPackMLMode_Auto.Enable := 0;
	MpPackMLMode_SemiAuto.Enable := 0;
	MpPackMLMode_Manual.Enable := 0;

	MpPackMLCore_0();
	MpPackMLMode_Auto();
	MpPackMLMode_SemiAuto();
	MpPackMLMode_Manual();

END_PROGRAM
```

### Program Logical/PackML/PackML_Auto (IEC)

#### Stopping.st
```iecst
ACTION Stopping:
	IF MpPackMLStateIsActive(gPackMLCore,
		mpPACKML_STATE_STOPPING,
		1) THEN

		PackML_State := 'STOPPING';

		//STOP EVERYTHING
		MpRoboArm6Axis_0.Stop := TRUE;
		IF NOT MpRoboArm6Axis_0.InMotion THEN
				MpRoboArm6Axis_0.Stop := FALSE;
			MpRoboArm6Axis_0.Power := FALSE;
			diStop := 0;

		//	IF NOT MpRoboArm6Axis_0.InMotion AND (NOT MpRoboArm6Axis_0.PowerOn) THEN

				MpPackMLStateComplete(gPackMLCore, 1);
		//	END_IF;

	END_IF;

	END_IF

END_ACTION
```

#### Starting.st
```iecst
ACTION Starting:

	IF MpPackMLStateIsActive(gPackMLCore,
		mpPACKML_STATE_STARTING,
		1) THEN

		MpPackMLMode_Auto.Start := 0;

		PackML_State := 'STARTING';

		Camera_0.ImageAcq := 0;

		DetectedSquares := 0;
		DetectedScrew := 0;
		DetectedScrewWasher := 0;
		DetectedWrench := 0;

		FOR i := 0 TO 13 DO
			//SQUARES DETECTION
			gSquareArray[Camera_0.ModelNumArray[i]-1] := Camera_0.PixelCntSquareArray[i] < PixelRange_0.HolderLimit;
			gIsPosGood[Camera_0.ModelNumArray[i]-1] := Camera_0.PixelCntSquareArray[i] < PixelRange_0.HolderLimit;
			IF Camera_0.PixelCntSquareArray[i] < PixelRange_0.HolderLimit THEN
				DetectedSquares := DetectedSquares + 1;
			END_IF

			IF Camera_0.PixelCntSquareArray[i] < 50 THEN
				//NOTHING
				gActPos[Camera_0.ModelNumArray[i]-1] := 0;
				gElementsArray[Camera_0.ModelNumArray[i]-1] := 0;
				DetectedScrew := 0;
				DetectedScrewWasher := 0;
				DetectedWrench := 0;
			ELSIF Camera_0.PixelCntSquareArray[i] < PixelRange_0.ScrewLimit THEN
				//SCREW
				gActPos[Camera_0.ModelNumArray[i]-1] := 1;
				gElementsArray[Camera_0.ModelNumArray[i]-1] := 1;
				DetectedScrew := DetectedScrew + 1;
			ELSIF Camera_0.PixelCntSquareArray[i] < PixelRange_0.WasherBoltLimit THEN
				//WASHER BOLT
				gActPos[Camera_0.ModelNumArray[i]-1] := 2;
				gElementsArray[Camera_0.ModelNumArray[i]-1] := 2;
				DetectedScrewWasher := DetectedScrewWasher + 1;
			ELSIF Camera_0.PixelCntSquareArray[i] < PixelRange_0.WrenchLimit THEN
				//WRENCH
				gActPos[Camera_0.ModelNumArray[i]-1] := 4;
				gElementsArray[Camera_0.ModelNumArray[i]-1] := 4;
				DetectedWrench := DetectedWrench + 1;
			ELSE
				gActPos[Camera_0.ModelNumArray[i]-1] := 0;
				gElementsArray[Camera_0.ModelNumArray[i]-1] := 0;
				DetectedScrew := 0;
				DetectedScrewWasher := 0;
				DetectedWrench := 0;
			END_IF;

		END_FOR;

		CASE Step OF
			ROBOTCTRL_CHECK: 	//checking if aim targets are available

				AimIsGood:=TRUE;
				FOR x:=0  TO SizeOfArray DO
					pom[0]:=1;
					IF gAimPos[x]>0 THEN
						pom[1]:=1;
						IF (gIsPosGood[x]=FALSE) THEN
							pom[2]:=1;
							Step:=ROBOTCTRL_ERROR_WRONG_AIM;
							Step_State := 'ERROR_WRONG_AIM';
							AimIsGood:=0;
						END_IF;
					END_IF;
				END_FOR;
				IF AimIsGood=TRUE THEN
					y:=0;
					Step:=ROBOTCTRL_CALCULATE;
					Step_State := 'CALCULATE';
					Camera_0.diTrigger := 0;
					MpPackMLStateComplete(gPackMLCore, 1);
				END_IF;

			ROBOTCTRL_ERROR_WRONG_AIM:
				//handling wrong target error
				doVisError:=TRUE;
				IF diAck THEN
					doVisError:=FALSE;

					Step:=ROBOTCTRL_CHECK;
					Step_State := 'CHECK';
				END_IF;

		END_CASE;

	END_IF
END_ACTION
```

#### Execute.st
```iecst
//   General conception of this code
//  assainging binary values to each object
//	screw      -001 - 1
//  screw pad  -010 - 2
//  wrench     -100 - 4
//  therefore we can assing to gAimPose table values from 0-7 ( sum must equal 7) in order to
//  easly differentiate what kind of object we need to move into aim pose.
//  for example if we see 6 -> 110 we know that we have to move screw pad and wrench to this pose
//
//  order of moves is defined by order of numbers in Index

ACTION Execute:
	IF MpPackMLStateIsActive(gPackMLCore,
		mpPACKML_STATE_EXECUTE,
		1) THEN

		PackML_State := 'EXECUTE';

		CASE Step OF
			ROBOTCTRL_CALCULATE:
				//blocks which can be used as buffor
				FOR x:=0 TO SizeOfArray DO
					IF  gActPos[x]=0 AND gIsPosGood[x]=TRUE THEN
						gPosBuffor[x]:=TRUE;
					END_IF;
				END_FOR;

				IF gSwapFlag THEN
					Step:=ROBOTCTRL_SWAP;
				ELSIF P1P2_Ok THEN
					Step:=ROBOTCTRL_IS_MOVE_NEEDED;
				ELSIF y<IndexSize THEN
					Step:=ROBOTCTRL_CALCULATE_P1;
				ELSE
					diStart:=FALSE;
					RoboParameters.ProgramName := 'HOME.st';
					MpRoboArm6Axis_0.MoveProgram:=1;
					IF MpRoboArm6Axis_0.MoveDone THEN
						MpRoboArm6Axis_0.MoveProgram:=FALSE;
						MpPackMLStateComplete(gPackMLCore, 1);
					END_IF

				END_IF;

			ROBOTCTRL_CALCULATE_P1:
				//assigning values to P1 and P1up
				FOR x:=0  TO SizeOfArray DO
					IF gActPos[x]=Index[y] THEN
						P1.Orient.Angle1:=gRobPos[x].Orient.Angle1;
						P1.Orient.Angle2:=gRobPos[x].Orient.Angle2;
						P1.Orient.Angle3:=gRobPos[x].Orient.Angle3;
						P1.Pos.X:=gRobPos[x].Pos.X;
						P1.Pos.Y:=gRobPos[x].Pos.Y;
						P1.Pos.Z:=gRobPos[x].Pos.Z;
						P1up.Orient.Angle1:=gRobPos[x].Orient.Angle1;
						P1up.Orient.Angle2:=gRobPos[x].Orient.Angle2;
						P1up.Orient.Angle3:=gRobPos[x].Orient.Angle3;
						P1up.Pos.X:=gRobPos[x].Pos.X;
						P1up.Pos.Y:=gRobPos[x].Pos.Y;
						P1up.Pos.Z:=gRobPos[x].Pos.Z+50;
					END_IF;
				END_FOR;
				Step:=ROBOTCTRL_CALCULATE_P2;
				Step_State := 'CALCULATE_P2';

			ROBOTCTRL_CALCULATE_P2:
				FOR x:=0 TO SizeOfArray DO
					//copig values
					gAimPos1[x]:=gAimPos[x];
				END_FOR;
				FOR x:=0 TO SizeOfArray DO
					//reseting maps
					Aim1[x]:=FALSE;
					Aim2[x]:=FALSE;
					Aim4[x]:=FALSE;
				END_FOR;
				//Creating maps conteining positions of each element
				//by substracting corresponding value of element
				//AND checing IF its greater OR equal TO zero
				FOR z:=0 TO IndexSize DO
					IF Index[z]=4 THEN
						FOR x:=0 TO SizeOfArray DO
							IF((gAimPos1[x]-4)>=0) THEN
								gAimPos1[x]:=gAimPos1[x]-4;
								Aim4[x]:=TRUE;
							END_IF;
						END_FOR;
					END_IF;
				END_FOR;

				FOR z:=0 TO IndexSize DO
					IF Index[z]=2 THEN
						FOR x:=0 TO SizeOfArray DO
							IF((gAimPos1[x]-2)>=0) THEN
								gAimPos1[x]:=gAimPos1[x]-2;
								Aim2[x]:=TRUE;
							END_IF;
						END_FOR;
					END_IF;
				END_FOR;

				FOR z:=0 TO IndexSize DO
					IF Index[z]=1 THEN
						FOR x:=0 TO SizeOfArray DO
							IF((gAimPos1[x]-1)>=0) THEN
								gAimPos1[x]:=gAimPos1[x]-1;
									Aim1[x]:=TRUE;
								END_IF;
							END_FOR;
						END_IF;
					END_FOR;

					//assigning values to P2 and P2up
				IF Index[y]=4 THEN
					//moving in order defined in Index
						FOR x:=0  TO SizeOfArray DO
							IF Aim4[x]=TRUE THEN
								P2.Orient.Angle1:=gRobPos[x].Orient.Angle1;
								P2.Orient.Angle2:=gRobPos[x].Orient.Angle2;
								P2.Orient.Angle3:=gRobPos[x].Orient.Angle3;
								P2.Pos.X:=gRobPos[x].Pos.X;
								P2.Pos.Y:=gRobPos[x].Pos.Y;
								P2.Pos.Z:=gRobPos[x].Pos.Z;
								P2up.Orient.Angle1:=gRobPos[x].Orient.Angle1;
								P2up.Orient.Angle2:=gRobPos[x].Orient.Angle2;
								P2up.Orient.Angle3:=gRobPos[x].Orient.Angle3;
								P2up.Pos.X:=gRobPos[x].Pos.X;
								P2up.Pos.Y:=gRobPos[x].Pos.Y;
								P2up.Pos.Z:=gRobPos[x].Pos.Z+50;
								END_IF;
							END_FOR;
						ELSIF Index[y]=2 THEN
						FOR x:=0  TO SizeOfArray DO
							IF Aim2[x]=TRUE THEN
								P2.Orient.Angle1:=gRobPos[x].Orient.Angle1;
								P2.Orient.Angle2:=gRobPos[x].Orient.Angle2;
								P2.Orient.Angle3:=gRobPos[x].Orient.Angle3;
								P2.Pos.X:=gRobPos[x].Pos.X;
								P2.Pos.Y:=gRobPos[x].Pos.Y;
								P2.Pos.Z:=gRobPos[x].Pos.Z;
								P2up.Orient.Angle1:=gRobPos[x].Orient.Angle1;
								P2up.Orient.Angle2:=gRobPos[x].Orient.Angle2;
								P2up.Orient.Angle3:=gRobPos[x].Orient.Angle3;
								P2up.Pos.X:=gRobPos[x].Pos.X;
								P2up.Pos.Y:=gRobPos[x].Pos.Y;
								P2up.Pos.Z:=gRobPos[x].Pos.Z+50;
							END_IF;
						END_FOR;
					ELSIF Index[y]=1 THEN
						FOR x:=0  TO SizeOfArray DO
							IF Aim1[x]=TRUE THEN
								P2.Orient.Angle1:=gRobPos[x].Orient.Angle1;
								P2.Orient.Angle2:=gRobPos[x].Orient.Angle2;
								P2.Orient.Angle3:=gRobPos[x].Orient.Angle3;
								P2.Pos.X:=gRobPos[x].Pos.X;
								P2.Pos.Y:=gRobPos[x].Pos.Y;
								P2.Pos.Z:=gRobPos[x].Pos.Z;
								P2up.Orient.Angle1:=gRobPos[x].Orient.Angle1;
								P2up.Orient.Angle2:=gRobPos[x].Orient.Angle2;
								P2up.Orient.Angle3:=gRobPos[x].Orient.Angle3;
								P2up.Pos.X:=gRobPos[x].Pos.X;
								P2up.Pos.Y:=gRobPos[x].Pos.Y;
								P2up.Pos.Z:=gRobPos[x].Pos.Z+50;
							END_IF;
						END_FOR;
					END_IF;
					P1P2_Ok:=1; // this flag means that new P1 and new P2 have been assigned
					Step:=ROBOTCTRL_CALCULATE;

			ROBOTCTRL_IS_MOVE_NEEDED:
				//checking if actual and aim positions are not the same
				IF P1.Orient.Angle1=P2.Orient.Angle1 AND P1.Pos.X=P2.Pos.X AND P1.Orient.Angle2=P2.Orient.Angle2 AND P1.Pos.Y=P2.Pos.Y AND P1.Orient.Angle3=P2.Orient.Angle3 AND P1.Pos.Z=P2.Pos.Z THEN
					y:=y+1; // index of next object
					P1P2_Ok:=0; // ready to assign new values to p1 p1up p2 p2up
					Step:=ROBOTCTRL_CALCULATE; // next assigning procedure with new object
					Step_State := 'CALCULATE';
				ELSE
					Step_State := 'MOVE';
					Step:=ROBOTCTRL_MOVE;   // going to move command
				END_IF;

			ROBOTCTRL_MOVE:
				IF cmdInterrupt OR MpRoboArm6Axis_0.MoveInterrupted THEN
					cmdInterrupt := FALSE;
					Step:=ROBOTCTRL_INTERRUPT;
					Step_State := 'INTERRUPT';
					MpPackMLMode_Auto.Hold := 1;
				END_IF;

				//executing move procedure
				MpRoboArm6Axis_0.MoveProgram:=1;
				IF MpRoboArm6Axis_0.MoveDone THEN
					//restarting assigning procedure with new object after finishing move
					MpRoboArm6Axis_0.MoveProgram:=0;
					y:=y+1;
					P1P2_Ok:=0;
					Step:=ROBOTCTRL_CALCULATE;
					Step_State := 'CALCULATE';

				END_IF

			ROBOTCTRL_SWAP:
				gSwapFlag:=FALSE;
				HelpfulInt:=0;
				FOR x:=0 TO SizeOfArray DO
					IF gSwapMap[x] THEN
						gSwapPoses[HelpfulInt].Orient.Angle1:=gRobPos[x].Orient.Angle1;
						gSwapPoses[HelpfulInt].Orient.Angle2:=gRobPos[x].Orient.Angle2;
						gSwapPoses[HelpfulInt].Orient.Angle3:=gRobPos[x].Orient.Angle3;
						gSwapPoses[HelpfulInt].Pos.X:=gRobPos[x].Pos.X;
						gSwapPoses[HelpfulInt].Pos.Y:=gRobPos[x].Pos.Y;
						gSwapPoses[HelpfulInt].Pos.Z:=gRobPos[x].Pos.Z;
						HelpfulInt:=HelpfulInt + 1;
					END_IF
				END_FOR;
				//gSwapMap should only have 2 values equal to TRUE therefore HelpfulInt should equal to 2
				//but just in case it is better to assign 2 to HelpfulInt
				HelpfulInt:=2;

				FOR x:=0 TO SizeOfArray DO
					IF gPosBuffor[x] THEN
						gSwapPoses[HelpfulInt].Orient.Angle1:=gRobPos[x].Orient.Angle1;
						gSwapPoses[HelpfulInt].Orient.Angle2:=gRobPos[x].Orient.Angle2;
						gSwapPoses[HelpfulInt].Orient.Angle3:=gRobPos[x].Orient.Angle3;
						gSwapPoses[HelpfulInt].Pos.X:=gRobPos[x].Pos.X;
						gSwapPoses[HelpfulInt].Pos.Y:=gRobPos[x].Pos.Y;
						gSwapPoses[HelpfulInt].Pos.Z:=gRobPos[x].Pos.Z;
						EXIT;
					END_IF
				END_FOR;

				FOR x:=0 TO SizeOfArray DO
					gSwapMap[x]:=FALSE;
				END_FOR;
				Step:=ROBOTCTRL_SWAP_MOVE;

			ROBOTCTRL_SWAP_MOVE:
				//first move
				///////////////////////P1
				P1.Orient.Angle1:=gSwapPoses[0].Orient.Angle1;
				P1.Orient.Angle2:=gSwapPoses[0].Orient.Angle2;
				P1.Orient.Angle3:=gSwapPoses[0].Orient.Angle3;
				P1.Pos.X:=gSwapPoses[0].Pos.X;
				P1.Pos.Y:=gSwapPoses[0].Pos.Y;
				P1.Pos.Z:=gSwapPoses[0].Pos.Z;
				P1up.Orient.Angle1:=gSwapPoses[0].Orient.Angle1;
				P1up.Orient.Angle2:=gSwapPoses[0].Orient.Angle2;
				P1up.Orient.Angle3:=gSwapPoses[0].Orient.Angle3;
				P1up.Pos.X:=gSwapPoses[0].Pos.X;
				P1up.Pos.Y:=gSwapPoses[0].Pos.Y;
				P1up.Pos.Z:=gSwapPoses[0].Pos.Z+50;
				///////////////////////P2
				P2.Orient.Angle1:=gSwapPoses[2].Orient.Angle1;
				P2.Orient.Angle2:=gSwapPoses[2].Orient.Angle2;
				P2.Orient.Angle3:=gSwapPoses[2].Orient.Angle3;
				P2.Pos.X:=gSwapPoses[2].Pos.X;
				P2.Pos.Y:=gSwapPoses[2].Pos.Y;
				P2.Pos.Z:=gSwapPoses[2].Pos.Z;
				P2up.Orient.Angle1:=gSwapPoses[2].Orient.Angle1;
				P2up.Orient.Angle2:=gSwapPoses[2].Orient.Angle2;
				P2up.Orient.Angle3:=gSwapPoses[2].Orient.Angle3;
				P2up.Pos.X:=gSwapPoses[2].Pos.X;
				P2up.Pos.Y:=gSwapPoses[2].Pos.Y;
				P2up.Pos.Z:=gSwapPoses[2].Pos.Z+50;
				//////////////////////// command execute
				MpRoboArm6Axis_0.MoveProgram:=1;
				IF MpRoboArm6Axis_0.MoveDone THEN
					//second move
					MpRoboArm6Axis_0.MoveProgram:=0;
					///////////////////////P1
					P1.Orient.Angle1:=gSwapPoses[0].Orient.Angle1;
					P1.Orient.Angle2:=gSwapPoses[0].Orient.Angle2;
					P1.Orient.Angle3:=gSwapPoses[0].Orient.Angle3;
					P1.Pos.X:=gSwapPoses[0].Pos.X;
					P1.Pos.Y:=gSwapPoses[0].Pos.Y;
					P1.Pos.Z:=gSwapPoses[0].Pos.Z;
					P1up.Orient.Angle1:=gSwapPoses[0].Orient.Angle1;
					P1up.Orient.Angle2:=gSwapPoses[0].Orient.Angle2;
					P1up.Orient.Angle3:=gSwapPoses[0].Orient.Angle3;
					P1up.Pos.X:=gSwapPoses[0].Pos.X;
					P1up.Pos.Y:=gSwapPoses[0].Pos.Y;
					P1up.Pos.Z:=gSwapPoses[0].Pos.Z+50;
					///////////////////////P2
					P2.Orient.Angle1:=gSwapPoses[1].Orient.Angle1;
					P2.Orient.Angle2:=gSwapPoses[1].Orient.Angle2;
					P2.Orient.Angle3:=gSwapPoses[1].Orient.Angle3;
					P2.Pos.X:=gSwapPoses[1].Pos.X;
					P2.Pos.Y:=gSwapPoses[1].Pos.Y;
					P2.Pos.Z:=gSwapPoses[1].Pos.Z;
					P2up.Orient.Angle1:=gSwapPoses[1].Orient.Angle1;
					P2up.Orient.Angle2:=gSwapPoses[1].Orient.Angle2;
					P2up.Orient.Angle3:=gSwapPoses[1].Orient.Angle3;
					P2up.Pos.X:=gSwapPoses[1].Pos.X;
					P2up.Pos.Y:=gSwapPoses[1].Pos.Y;
					P2up.Pos.Z:=gSwapPoses[1].Pos.Z+50;
					//////////////////////// command execute
					MpRoboArm6Axis_0.MoveProgram:=1;
					IF MpRoboArm6Axis_0.MoveDone THEN
						//third move
						MpRoboArm6Axis_0.MoveProgram:=0;
						///////////////////////P1
						P1.Orient.Angle1:=gSwapPoses[2].Orient.Angle1;
						P1.Orient.Angle2:=gSwapPoses[2].Orient.Angle2;
						P1.Orient.Angle3:=gSwapPoses[2].Orient.Angle3;
						P1.Pos.X:=gSwapPoses[2].Pos.X;
						P1.Pos.Y:=gSwapPoses[2].Pos.Y;
						P1.Pos.Z:=gSwapPoses[2].Pos.Z;
						P1up.Orient.Angle1:=gSwapPoses[2].Orient.Angle1;
						P1up.Orient.Angle2:=gSwapPoses[2].Orient.Angle2;
						P1up.Orient.Angle3:=gSwapPoses[2].Orient.Angle3;
						P1up.Pos.X:=gSwapPoses[2].Pos.X;
						P1up.Pos.Y:=gSwapPoses[2].Pos.Y;
						P1up.Pos.Z:=gSwapPoses[2].Pos.Z+50;
						///////////////////////P2
						P2.Orient.Angle1:=gSwapPoses[0].Orient.Angle1;
						P2.Orient.Angle2:=gSwapPoses[0].Orient.Angle2;
						P2.Orient.Angle3:=gSwapPoses[0].Orient.Angle3;
						P2.Pos.X:=gSwapPoses[0].Pos.X;
						P2.Pos.Y:=gSwapPoses[0].Pos.Y;
						P2.Pos.Z:=gSwapPoses[0].Pos.Z;
						P2up.Orient.Angle1:=gSwapPoses[0].Orient.Angle1;
						P2up.Orient.Angle2:=gSwapPoses[0].Orient.Angle2;
						P2up.Orient.Angle3:=gSwapPoses[0].Orient.Angle3;
						P2up.Pos.X:=gSwapPoses[0].Pos.X;
						P2up.Pos.Y:=gSwapPoses[0].Pos.Y;
						P2up.Pos.Z:=gSwapPoses[0].Pos.Z+50;
						//////////////////////// command execute
						MpRoboArm6Axis_0.MoveProgram:=1;
					END_IF
				END_IF
		END_CASE;

	END_IF

END_ACTION
```

#### Completing.st
```iecst
ACTION Completing:
	IF MpPackMLStateIsActive(gPackMLCore,
		mpPACKML_STATE_COMPLETING,
		1) THEN
			PackML_State := 'COMPLETING';

			MpPackMLStateComplete(gPackMLCore, 1);

	END_IF

END_ACTION
```

#### Complete.st
```iecst
ACTION Complete:
	IF MpPackMLStateIsActive(gPackMLCore,
		mpPACKML_STATE_COMPLETE,
		1) THEN

		PackML_State := 'COMPLETE';

	//MpPackMLMode_Auto.Stop := 1;
		IF diReset THEN
			MpPackMLStateComplete(gPackMLCore, 1);
			MpPackMLMode_Auto.Reset := 1;
			Step := ROBOTCTRL_POWER;

			//			Step_State := 'POWER';

			END_IF;
	END_IF

END_ACTION
```

#### Main.st - Init, cyclic, exit code
```iecst
PROGRAM _INIT
	RestorePos;
	MpRoboArm6Axis_0.Enable := TRUE;

	MpRoboArm6Axis_0.Interrupt := 0;
	MpRoboArm6Axis_0.Continue := 0;

	MpRoboArm6Axis_0.Override  := 100.0;
	RoboParameters.CoordSystem := 0;
	RoboParameters.Velocity := 100;
	RoboParameters.Acceleration := 1000;
	RoboParameters.Deceleration := 1000;
	RoboParameters.ProgramName := 'Robotic.st';

END_PROGRAM

PROGRAM _CYCLIC
	Starting;
	Idle;
	Stopping;
	Resetting;
	Execute;
	Completing;
	Complete;
	Stopped;
	Holding;
	Held;
	Unhold;
	Aborted;
	Aborting;
	Clearing;

	P2up;
	P2 ;
	P1up ;
	P1 ;
	P0;
	HOME;
	PZ;
	A;
	doMagnet;
	MaxSpeed;
	LowSpeed;

	IF diAck THEN
		doVisError:=FALSE;

	END_IF;

	//throwing error
	IF MpRoboArm6Axis_0.Error THEN
//		Step := ROBOTCTRL_ERROR;
		MpPackMLMode_Auto.Abort := TRUE;
//		Step_State := 'ERROR';
	END_IF;

	IF diStop THEN
		MpRoboArm6Axis_0.Power := 0;
		MpPackMLMode_Auto.Stop := 1;
//		Step := ROBOTCTRL_POWER_OFF;
//		Step_State := 'POWER_OFF';
	END_IF

	MpPackMLCore_0;
	MpPackMLMode_Auto;

	diStop;
	diStart;
	diReset;
	diExecute;
	cmdContinue;

	diAuto;
	diSemiAuto;
	diManual;

	MpRoboArm6Axis_0.MpLink     := ADR(gAxesGroup_Racer3_1);
	MpRoboArm6Axis_0.Parameters := ADR(RoboParameters);
	MpRoboArm6Axis_0.Override := 100.0;
	MpRoboArm6Axis_0.Enable := TRUE;
	MpRoboArm6Axis_0();

END_PROGRAM

PROGRAM _EXIT

END_PROGRAM
```

### Program Logical/PackML/PackML_SemiAuto (IEC)

#### Main.st
```iecst
PROGRAM _INIT
	(* Insert code here *)

END_PROGRAM

PROGRAM _CYCLIC
	Starting;
	Idle;
	Stopping;
	Resetting;
	Execute;
	Completing;
	Complete;
	Stopped;

END_PROGRAM

PROGRAM _EXIT
	(* Insert code here *)

END_PROGRAM
```

### Program Logical/PackML/PackML_Manual (IEC)

#### Idle.st
```iecst
ACTION Idle:

END_ACTION
```

#### Resetting.st
```iecst
ACTION Resetting:

END_ACTION
```

### Variables.var
```iecst
VAR
	AimIsGood : BOOL := FALSE;
	cartezianVSjog : BOOL; (*Wybór miedzy sterowaniem we wspólrzednych wewnetrznych - 0 / zewnętrznych - 1 *)
	cmdContinue : BOOL;
	cmdInterrupt : BOOL;
	diAck : BOOL;
	diAuto : BOOL;
	diExecute : BOOL;
	diManual : BOOL;
	diReset : BOOL;
	diSemiAuto : BOOL;
	diStart : BOOL;
	diStop : BOOL;
END_VAR
VAR CONSTANT

	IndexSize : INT := 3;
END_VAR
VAR
	MpRoboArm6Axis_0 : MpRoboArm6Axis;
	P1P2_Ok : BOOL := FALSE;
	RoboParameters : MpRoboArm6AxisParType;
END_VAR
VAR CONSTANT
	SizeOfArray : INT := 13;
END_VAR
VAR
	Step : {REDUND_UNREPLICABLE} Step_typ := (0);
	VelocityQ : REAL;
	VelocityQ1 : REAL; (*Przypisanie predkosci do parametru 1 w zależnosci od wyboru wspólrzednych*)
	VelocityQ2 : REAL; (*Przypisanie predkosci do parametru 2 w zależnosci od wyboru wspólrzednych*)
	VelocityQ3 : REAL; (*Przypisanie predkosci do parametru 3 w zależnosci od wyboru wspólrzednych*)
	VelocityQ4 : REAL; (*Przypisanie predkosci do parametru 4 w zależnosci od wyboru wspólrzednych*)
	VelocityQ5 : REAL; (*Przypisanie predkosci do parametru 5 w zależnosci od wyboru wspólrzednych*)
	VelocityQ6 : REAL; (*Przypisanie predkosci do parametru 6 w zależnosci od wyboru wspólrzednych*)
	Step_State : STRING[80];
	PackML_State : STRING[80];
	VisionCalcDone : BOOL;
	x : INT := 0;
END_VAR
```

### Types.typ
```iecst
TYPE
	Step_typ :
		(
		ROBOTCTRL_DISABLED,
		ROBOTCTRL_POWER,
		ROBOTCTRL_WAIT_POWER,
		ROBOTCTRL_HOME,
		ROBOTCTRL_WAIT_HOME,
		ROBOTCTRL_READY,
		ROBOTCTRL_CALCULATE,
		ROBOTCTRL_CHECK,
		ROBOTCTRL_CALCULATE_P1,
		ROBOTCTRL_CALCULATE_P2,
		ROBOTCTRL_IS_MOVE_NEEDED,
		ROBOTCTRL_MOVE,
		ROBOTCTRL_ERROR_WRONG_AIM,
		ROBOTCTRL_ERROR,
		ROBOTCTRL_STOP,
		ROBOTCTRL_INTERRUPT,
		ROBOTCTRL_INTERRUPTING,
		ROBOTCTRL_CONTINUE,
		ROBOTCTRL_POWER_OFF,
		ROBOTCTRL_COMPLITE,
		ROBOTCTRL_SWAP,
			ROBOTCTRL_SWAP_MOVE
		);
END_TYPE
```

### Variables.var
```iecst
VAR
	clear : BOOL;
	MpRecipeXml_0 : MpRecipeXml;
	name2 : STRING[80];
	name : STRING[80];
	ScrewWasher : BOOL;
	Wrench : BOOL;
	Screw : BOOL;
	MpRecipeRegPar_0 : MpRecipeRegPar;
	ScrewPosible : BOOL;
	WrenchPosible : BOOL;
	ScrewWasherPosible : BOOL;
	i : INT;
	iFile : INT;
	MpFileManagerUI_R : MpFileManagerUI;
	MpFileMngSetup : MpFileManagerUISetupType;
	MpFileMngConnectR : MpFileManagerUIConnectType;
	tabInfo : TabInfo;
	messageType : STRING[80];
	tempString : STRING[200];
	tableConfig : STRING[200];
	testString : STRING[200] := '{"specRows": [ {"from":0, "to":3, "visible":true}, {"from":4, "to":49, "visible":false}]}';
	tableShowLimit : INT;
	PriorytetS : INT;
	PriorytetSW : INT;
	PriorytetW : INT;
	makeWarning : USINT;
END_VAR
```

Listed in the project but not available here: Logical/PackML/PackML_Auto/Types.typ, Logical/PackML/PackML_Auto/Stopped.st, Logical/PackML/PackML_Auto/Resetting.st, Logical/PackML/PackML_Auto/Idle.st, Logical/PackML/PackML_Auto/Holding.st, Logical/PackML/PackML_Auto/Held.st, Logical/PackML/PackML_Auto/Unhold.st, Logical/PackML/PackML_Auto/Aborting.st, Logical/PackML/PackML_Auto/Aborted.st, Logical/PackML/PackML_Auto/Clearing.st, Logical/PackML/PackML_Manual/Main.st, Logical/PackML/PackML_Manual/Types.typ, Logical/PackML/PackML_Manual/Variables.var, Logical/PackML/PackML_Manual/Starting.st, Logical/PackML/PackML_Manual/Stopping.st, Logical/PackML/PackML_Manual/Execute.st, Logical/PackML/PackML_Manual/Completing.st, Logical/PackML/PackML_Manual/Complete.st, Logical/PackML/PackML_Manual/Stopped.st
